LIN {X 0,Y 441.863,Z 860.022,A -85,B 0,C 180,E1 -9104.979,E2 -9104.979} C_VEL
LIN {X 0,Y 442.081,Z 852.631,A -85,B 0,C 180,E1 -9105.384,E2 -9105.384} C_VEL
LIN {X 0,Y 440.393,Z 839.206,A -85,B 0,C 180,E1 -9106.023,E2 -9106.023} C_VEL
LIN {X 0,Y 438.824,Z 827.47,A -85,B 0,C 180,E1 -9106.443,E2 -9106.443} C_VEL
LIN {X 0,Y 439.003,Z 818.523,A -85,B 0,C 180,E1 -9109.645,E2 -9109.645} C_VEL
LIN {X 0,Y 439.338,Z 809.24,A -85,B 0,C 180,E1 -9113.074,E2 -9113.074} C_VEL
LIN {X 0,Y 439.723,Z 800.458,A -85,B 0,C 180,E1 -9116.486,E2 -9116.486} C_VEL
LIN {X 0,Y 440.208,Z 792.815,A -85,B 0,C 180,E1 -9119.665,E2 -9119.665} C_VEL
LIN {X 0,Y 440.836,Z 785.884,A -85,B 0,C 180,E1 -9122.823,E2 -9122.823} C_VEL
LIN {X 0,Y 441.25,Z 781.634,A -85,B 0,C 180,E1 -9124.987,E2 -9124.987} C_VEL
LIN {X 0,Y 441.238,Z 777.8,A -85,B 0,C 180,E1 -9127.248,E2 -9127.248} C_VEL
LIN {X 0,Y 440.674,Z 774.022,A -85,B 0,C 180,E1 -9130.046,E2 -9130.046} C_VEL
LIN {X 0,Y 440.207,Z 771.332,A -85,B 0,C 180,E1 -9132.743,E2 -9132.743} C_VEL
LIN {X 0,Y 439.877,Z 769.661,A -85,B 0,C 180,E1 -9135.331,E2 -9135.331} C_VEL
LIN {X 0,Y 439.737,Z 768.806,A -85,B 0,C 180,E1 -9137.835,E2 -9137.835} C_VEL
LIN {X 0,Y 439.694,Z 768.625,A -85,B 0,C 180,E1 -9140.256,E2 -9140.256} C_VEL
LIN {X 0,Y 439.718,Z 769.039,A -85,B 0,C 180,E1 -9143.049,E2 -9143.049} C_VEL
LIN {X 0,Y 439.636,Z 770.08,A -85,B 0,C 180,E1 -9145.977,E2 -9145.977} C_VEL
LIN {X 0,Y 439.502,Z 771.14,A -85,B 0,C 180,E1 -9148.149,E2 -9148.149} C_VEL
LIN {X 0,Y 439.208,Z 773.033,A -85,B 0,C 180,E1 -9151.311,E2 -9151.311} C_VEL
LIN {X 0,Y 439.029,Z 775.128,A -85,B 0,C 180,E1 -9154.391,E2 -9154.391} C_VEL
LIN {X 0,Y 438.912,Z 777.387,A -85,B 0,C 180,E1 -9157.399,E2 -9157.399} C_VEL
LIN {X 0,Y 438.78,Z 779.764,A -85,B 0,C 180,E1 -9160.344,E2 -9160.344} C_VEL
LIN {X 0,Y 438.668,Z 782.635,A -85,B 0,C 180,E1 -9163.693,E2 -9163.693} C_VEL
LIN {X 0,Y 442.001,Z 795.437,A -85,B 0,C 180,E1 -9164.317,E2 -9164.317} C_VEL
LIN {X 0,Y 442.761,Z 800.41,A -85,B 0,C 180,E1 -9164.58,E2 -9164.58} C_VEL
LIN {X 0,Y 442.269,Z 812.861,A -85,B 0,C 180,E1 -9165.27,E2 -9165.27} C_VEL
LIN {X 0,Y 441.715,Z 823.88,A -85,B 0,C 180,E1 -9166.062,E2 -9166.062} C_VEL
LIN {X 0,Y 441.095,Z 835.387,A -85,B 0,C 180,E1 -9167.11,E2 -9167.11} C_VEL
LIN {X 0,Y 440.405,Z 845.56,A -85,B 0,C 180,E1 -9168.259,E2 -9168.259} C_VEL
LIN {X 0,Y 439.861,Z 855.273,A -85,B 0,C 180,E1 -9169.644,E2 -9169.644} C_VEL
LIN {X 0,Y 439.359,Z 863.095,A -85,B 0,C 180,E1 -9171.027,E2 -9171.027} C_VEL
LIN {X 0,Y 439.018,Z 868.375,A -85,B 0,C 180,E1 -9172.179,E2 -9172.179} C_VEL
LIN {X 0,Y 438.847,Z 873.537,A -85,B 0,C 180,E1 -9173.563,E2 -9173.563} C_VEL
LIN {X 0,Y 438.558,Z 877.539,A -85,B 0,C 180,E1 -9174.943,E2 -9174.943} C_VEL
LIN {X 0,Y 438.53,Z 880.466,A -85,B 0,C 180,E1 -9176.324,E2 -9176.324} C_VEL
LIN {X 0,Y 438.434,Z 881.88,A -85,B 0,C 180,E1 -9177.243,E2 -9177.243} C_VEL
LIN {X 0,Y 438.451,Z 882.856,A -85,B 0,C 180,E1 -9178.162,E2 -9178.162} C_VEL
LIN {X 0,Y 438.338,Z 883.651,A -85,B 0,C 180,E1 -9179.999,E2 -9179.999} C_VEL
LIN {X 0,Y 438.367,Z 883.419,A -85,B 0,C 180,E1 -9180.918,E2 -9180.918} C_VEL
LIN {X 0,Y 438.429,Z 882.781,A -85,B 0,C 180,E1 -9181.836,E2 -9181.836} C_VEL
LIN {X 0,Y 438.405,Z 881.756,A -85,B 0,C 180,E1 -9182.756,E2 -9182.756} C_VEL
LIN {X 0,Y 438.516,Z 880.324,A -85,B 0,C 180,E1 -9183.675,E2 -9183.675} C_VEL
LIN {X 0,Y 438.493,Z 877.344,A -85,B 0,C 180,E1 -9185.056,E2 -9185.056} C_VEL
LIN {X 0,Y 438.765,Z 873.305,A -85,B 0,C 180,E1 -9186.437,E2 -9186.437} C_VEL
LIN {X 0,Y 438.997,Z 867.096,A -85,B 0,C 180,E1 -9188.052,E2 -9188.052} C_VEL
LIN {X 0,Y 439.42,Z 860.319,A -85,B 0,C 180,E1 -9189.434,E2 -9189.434} C_VEL
LIN {X 0,Y 439.925,Z 851.912,A -85,B 0,C 180,E1 -9190.818,E2 -9190.818} C_VEL
LIN {X 0,Y 440.418,Z 843.258,A -85,B 0,C 180,E1 -9191.972,E2 -9191.972} C_VEL
LIN {X 0,Y 441.03,Z 833.231,A -85,B 0,C 180,E1 -9193.064,E2 -9193.064} C_VEL
LIN {X 0,Y 441.548,Z 822.138,A -85,B 0,C 180,E1 -9194.047,E2 -9194.047} C_VEL
LIN {X 0,Y 442.104,Z 810.557,A -85,B 0,C 180,E1 -9194.852,E2 -9194.852} C_VEL
LIN {X 0,Y 442.538,Z 799.996,A -85,B 0,C 180,E1 -9195.426,E2 -9195.426} C_VEL
LIN {X 0,Y 440.768,Z 790.018,A -85,B 0,C 180,E1 -9195.922,E2 -9195.922} C_VEL
LIN {X 0,Y 438.433,Z 780.272,A -85,B 0,C 180,E1 -9196.344,E2 -9196.344} C_VEL
LIN {X 0,Y 438.467,Z 776.8,A -85,B 0,C 180,E1 -9199.669,E2 -9199.669} C_VEL
LIN {X 0,Y 438.535,Z 773.779,A -85,B 0,C 180,E1 -9202.619,E2 -9202.619} C_VEL
LIN {X 0,Y 438.643,Z 770.171,A -85,B 0,C 180,E1 -9206.202,E2 -9206.202} C_VEL
LIN {X 0,Y 438.702,Z 766.841,A -85,B 0,C 180,E1 -9209.775,E2 -9209.775} C_VEL
LIN {X 0,Y 439.093,Z 766.791,A -85,B 0,C 180,E1 -9212.968,E2 -9212.968} C_VEL
LIN {X 0,Y 439.308,Z 766.762,A -85,B 0,C 180,E1 -9215.324,E2 -9215.324} C_VEL
LIN {X 0,Y 439.373,Z 766.754,A -85,B 0,C 180,E1 -9218.594,E2 -9218.594} C_VEL
LIN {X 0,Y 439.384,Z 766.754,A -85,B 0,C 180,E1 -9221.256,E2 -9221.256} C_VEL
LIN {X 0,Y 439.396,Z 766.751,A -85,B 0,C 180,E1 -9224.728,E2 -9224.728} C_VEL
LIN {X 0,Y 439.39,Z 766.752,A -85,B 0,C 180,E1 -9227.795,E2 -9227.795} C_VEL
LIN {X 0,Y 439.404,Z 766.749,A -85,B 0,C 180,E1 -9230.225,E2 -9230.225} C_VEL
LIN {X 0,Y 439.366,Z 766.755,A -85,B 0,C 180,E1 -9233.712,E2 -9233.712} C_VEL
LIN {X 0,Y 439.364,Z 766.756,A -85,B 0,C 180,E1 -9237.053,E2 -9237.053} C_VEL
LIN {X 0,Y 439.369,Z 766.754,A -85,B 0,C 180,E1 -9240.273,E2 -9240.273} C_VEL
LIN {X 0,Y 439.373,Z 766.757,A -85,B 0,C 180,E1 -9243.392,E2 -9243.392} C_VEL
LIN {X 0,Y 439.373,Z 766.752,A -85,B 0,C 180,E1 -9246.429,E2 -9246.429} C_VEL
LIN {X 0,Y 439.379,Z 766.755,A -85,B 0,C 180,E1 -9249.397,E2 -9249.397} C_VEL
LIN {X 0,Y 439.395,Z 766.75,A -85,B 0,C 180,E1 -9252.308,E2 -9252.308} C_VEL
LIN {X 0,Y 439.437,Z 766.745,A -85,B 0,C 180,E1 -9255.174,E2 -9255.174} C_VEL
LIN {X 0,Y 439.473,Z 766.743,A -85,B 0,C 180,E1 -9258.001,E2 -9258.001} C_VEL
LIN {X 0,Y 439.491,Z 766.742,A -85,B 0,C 180,E1 -9261.725,E2 -9261.725} C_VEL
LIN {X 0,Y 439.586,Z 766.725,A -85,B 0,C 180,E1 -9264.495,E2 -9264.495} C_VEL
LIN {X 0,Y 439.516,Z 766.732,A -85,B 0,C 180,E1 -9266.988,E2 -9266.988} C_VEL
LIN {X 0,Y 439.304,Z 766.763,A -85,B 0,C 180,E1 -9267.499,E2 -9267.499} C_VEL
LIN {X 0,Y 438.003,Z 766.928,A -85,B 0,C 180,E1 -9268.254,E2 -9268.254} C_VEL
LIN {X 0,Y 433.58,Z 767.48,A -85,B 0,C 180,E1 -9269.996,E2 -9269.996} C_VEL
LIN {X 0,Y 432.529,Z 767.604,A -85,B 0,C 180,E1 -9270.773,E2 -9270.773} C_VEL
LIN {X 0,Y 432.464,Z 767.611,A -85,B 0,C 180,E1 -9271.036,E2 -9271.036} C_VEL
LIN {X 0,Y 432.543,Z 767.601,A -85,B 0,C 180,E1 -9272.794,E2 -9272.794} C_VEL
LIN {X 0,Y 432.503,Z 767.609,A -85,B 0,C 180,E1 -9276.531,E2 -9276.531} C_VEL
LIN {X 0,Y 432.408,Z 767.618,A -85,B 0,C 180,E1 -9279.354,E2 -9279.354} C_VEL
LIN {X 0,Y 432.421,Z 767.618,A -85,B 0,C 180,E1 -9282.803,E2 -9282.803} C_VEL
LIN {X 0,Y 432.402,Z 767.625,A -85,B 0,C 180,E1 -9286.478,E2 -9286.478} C_VEL
LIN {X 0,Y 432.329,Z 767.63,A -85,B 0,C 180,E1 -9289.961,E2 -9289.961} C_VEL
LIN {X 0,Y 432.307,Z 767.633,A -85,B 0,C 180,E1 -9292.965,E2 -9292.965} C_VEL
LIN {X 0,Y 432.325,Z 767.631,A -85,B 0,C 180,E1 -9295.003,E2 -9295.003} C_VEL
LIN {X 0,Y 432.334,Z 767.63,A -85,B 0,C 180,E1 -9298.127,E2 -9298.127} C_VEL
LIN {X 0,Y 432.312,Z 767.632,A -85,B 0,C 180,E1 -9301.347,E2 -9301.347} C_VEL
LIN {X 0,Y 432.33,Z 767.634,A -85,B 0,C 180,E1 -9304.678,E2 -9304.678} C_VEL
LIN {X 0,Y 432.329,Z 767.63,A -85,B 0,C 180,E1 -9308.151,E2 -9308.151} C_VEL
LIN {X 0,Y 432.326,Z 767.631,A -85,B 0,C 180,E1 -9311.603,E2 -9311.603} C_VEL
LIN {X 0,Y 432.328,Z 767.631,A -85,B 0,C 180,E1 -9314.348,E2 -9314.348} C_VEL
LIN {X 0,Y 432.315,Z 767.637,A -85,B 0,C 180,E1 -9317.017,E2 -9317.017} C_VEL
LIN {X 0,Y 432.329,Z 767.631,A -85,B 0,C 180,E1 -9319.822,E2 -9319.822} C_VEL
LIN {X 0,Y 432.295,Z 767.638,A -85,B 0,C 180,E1 -9323.022,E2 -9323.022} C_VEL
LIN {X 0,Y 432.168,Z 767.654,A -85,B 0,C 180,E1 -9326.035,E2 -9326.035} C_VEL
LIN {X 0,Y 431.864,Z 767.69,A -85,B 0,C 180,E1 -9328.618,E2 -9328.618} C_VEL
LIN {X 0,Y 431.471,Z 767.743,A -85,B 0,C 180,E1 -9331.813,E2 -9331.813} C_VEL
LIN {X 0,Y 431.514,Z 769.976,A -85,B 0,C 180,E1 -9333.914,E2 -9333.914} C_VEL
LIN {X 0,Y 431.405,Z 773.326,A -85,B 0,C 180,E1 -9336.986,E2 -9336.986} C_VEL
LIN {X 0,Y 431.382,Z 776.555,A -85,B 0,C 180,E1 -9339.995,E2 -9339.995} C_VEL
LIN {X 0,Y 431.355,Z 780.414,A -85,B 0,C 180,E1 -9343.533,E2 -9343.533} C_VEL
LIN {X 0,Y 434.362,Z 793.612,A -85,B 0,C 180,E1 -9344.097,E2 -9344.097} C_VEL
LIN {X 0,Y 435.602,Z 801.29,A -85,B 0,C 180,E1 -9344.504,E2 -9344.504} C_VEL
LIN {X 0,Y 435.12,Z 812.506,A -85,B 0,C 180,E1 -9345.144,E2 -9345.144} C_VEL
LIN {X 0,Y 434.523,Z 823.742,A -85,B 0,C 180,E1 -9345.96,E2 -9345.96} C_VEL
LIN {X 0,Y 433.987,Z 835.113,A -85,B 0,C 180,E1 -9347.016,E2 -9347.016} C_VEL
LIN {X 0,Y 433.335,Z 844.381,A -85,B 0,C 180,E1 -9348.067,E2 -9348.067} C_VEL
LIN {X 0,Y 432.861,Z 852.9,A -85,B 0,C 180,E1 -9349.24,E2 -9349.24} C_VEL
LIN {X 0,Y 432.333,Z 861.184,A -85,B 0,C 180,E1 -9350.646,E2 -9350.646} C_VEL
LIN {X 0,Y 431.905,Z 867.856,A -85,B 0,C 180,E1 -9352.051,E2 -9352.051} C_VEL
LIN {X 0,Y 431.699,Z 873.179,A -85,B 0,C 180,E1 -9353.457,E2 -9353.457} C_VEL
LIN {X 0,Y 431.44,Z 877.326,A -85,B 0,C 180,E1 -9354.861,E2 -9354.861} C_VEL
LIN {X 0,Y 431.45,Z 880.397,A -85,B 0,C 180,E1 -9356.265,E2 -9356.265} C_VEL
LIN {X 0,Y 431.33,Z 881.916,A -85,B 0,C 180,E1 -9357.199,E2 -9357.199} C_VEL
LIN {X 0,Y 431.328,Z 882.978,A -85,B 0,C 180,E1 -9358.133,E2 -9358.133} C_VEL
LIN {X 0,Y 431.308,Z 883.654,A -85,B 0,C 180,E1 -9359.067,E2 -9359.067} C_VEL
LIN {X 0,Y 431.277,Z 883.943,A -85,B 0,C 180,E1 -9360.001,E2 -9360.001} C_VEL
LIN {X 0,Y 431.309,Z 883.789,A -85,B 0,C 180,E1 -9360.935,E2 -9360.935} C_VEL
LIN {X 0,Y 431.345,Z 883.232,A -85,B 0,C 180,E1 -9361.868,E2 -9361.868} C_VEL
LIN {X 0,Y 431.348,Z 882.291,A -85,B 0,C 180,E1 -9362.803,E2 -9362.803} C_VEL
LIN {X 0,Y 431.466,Z 880.928,A -85,B 0,C 180,E1 -9363.737,E2 -9363.737} C_VEL
LIN {X 0,Y 431.467,Z 878.071,A -85,B 0,C 180,E1 -9365.141,E2 -9365.141} C_VEL
LIN {X 0,Y 431.78,Z 874.144,A -85,B 0,C 180,E1 -9366.543,E2 -9366.543} C_VEL
LIN {X 0,Y 431.987,Z 869.057,A -85,B 0,C 180,E1 -9367.95,E2 -9367.95} C_VEL
LIN {X 0,Y 432.396,Z 862.638,A -85,B 0,C 180,E1 -9369.355,E2 -9369.355} C_VEL
LIN {X 0,Y 432.955,Z 854.665,A -85,B 0,C 180,E1 -9370.76,E2 -9370.76} C_VEL
LIN {X 0,Y 433.454,Z 846.49,A -85,B 0,C 180,E1 -9371.932,E2 -9371.932} C_VEL
LIN {X 0,Y 434.143,Z 836.441,A -85,B 0,C 180,E1 -9373.1,E2 -9373.1} C_VEL
LIN {X 0,Y 434.685,Z 825.348,A -85,B 0,C 180,E1 -9374.156,E2 -9374.156} C_VEL
LIN {X 0,Y 435.439,Z 812.658,A -85,B 0,C 180,E1 -9375.086,E2 -9375.086} C_VEL
LIN {X 0,Y 435.939,Z 801.427,A -85,B 0,C 180,E1 -9375.727,E2 -9375.727} C_VEL
LIN {X 0,Y 434.163,Z 791.998,A -85,B 0,C 180,E1 -9376.237,E2 -9376.237} C_VEL
LIN {X 0,Y 431.559,Z 782.504,A -85,B 0,C 180,E1 -9376.694,E2 -9376.694} C_VEL
LIN {X 0,Y 431.548,Z 778.931,A -85,B 0,C 180,E1 -9379.999,E2 -9379.999} C_VEL
LIN {X 0,Y 431.615,Z 775.631,A -85,B 0,C 180,E1 -9383.005,E2 -9383.005} C_VEL
LIN {X 0,Y 431.67,Z 772.181,A -85,B 0,C 180,E1 -9386.078,E2 -9386.078} C_VEL
LIN {X 0,Y 431.645,Z 768.422,A -85,B 0,C 180,E1 -9389.24,E2 -9389.24} C_VEL
LIN {X 0,Y 431.711,Z 767.713,A -85,B 0,C 180,E1 -9390.366,E2 -9390.366} C_VEL
LIN {X 0,Y 432.113,Z 767.663,A -85,B 0,C 180,E1 -9393.573,E2 -9393.573} C_VEL
LIN {X 0,Y 432.273,Z 767.639,A -85,B 0,C 180,E1 -9395.825,E2 -9395.825} C_VEL
LIN {X 0,Y 432.337,Z 767.632,A -85,B 0,C 180,E1 -9398.713,E2 -9398.713} C_VEL
LIN {X 0,Y 432.329,Z 767.631,A -85,B 0,C 180,E1 -9401.799,E2 -9401.799} C_VEL
LIN {X 0,Y 432.338,Z 767.631,A -85,B 0,C 180,E1 -9404.348,E2 -9404.348} C_VEL
LIN {X 0,Y 432.382,Z 767.68,A -85,B 0,C 180,E1 -9407.817,E2 -9407.817} C_VEL
LIN {X 0,Y 433.57,Z 774.337,A -85,B 0,C 180,E1 -9411.084,E2 -9411.084} C_VEL
LIN {X 0,Y 434.286,Z 778.889,A -85,B 0,C 180,E1 -9413.218,E2 -9413.218} C_VEL
LIN {X 0,Y 434.361,Z 782.778,A -85,B 0,C 180,E1 -9414.943,E2 -9414.943} C_VEL
LIN {X 0,Y 433.81,Z 790.498,A -85,B 0,C 180,E1 -9418.229,E2 -9418.229} C_VEL
LIN {X 0,Y 433.312,Z 797.589,A -85,B 0,C 180,E1 -9421.146,E2 -9421.146} C_VEL
LIN {X 0,Y 432.793,Z 805.999,A -85,B 0,C 180,E1 -9424.512,E2 -9424.512} C_VEL
LIN {X 0,Y 432.309,Z 815.073,A -85,B 0,C 180,E1 -9428.043,E2 -9428.043} C_VEL
LIN {X 0,Y 432,Z 822.85,A -85,B 0,C 180,E1 -9431.012,E2 -9431.012} C_VEL
LIN {X 0,Y 431.769,Z 829.127,A -85,B 0,C 180,E1 -9433.372,E2 -9433.372} C_VEL
LIN {X 0,Y 433.924,Z 843.779,A -85,B 0,C 180,E1 -9433.915,E2 -9433.915} C_VEL
LIN {X 0,Y 435.32,Z 855.22,A -85,B 0,C 180,E1 -9434.491,E2 -9434.491} C_VEL
LIN {X 0,Y 434.594,Z 867.79,A -85,B 0,C 180,E1 -9435.244,E2 -9435.244} C_VEL
LIN {X 0,Y 433.967,Z 879.201,A -85,B 0,C 180,E1 -9436.128,E2 -9436.128} C_VEL
LIN {X 0,Y 433.304,Z 890.451,A -85,B 0,C 180,E1 -9437.233,E2 -9437.233} C_VEL
LIN {X 0,Y 432.665,Z 901.007,A -85,B 0,C 180,E1 -9438.522,E2 -9438.522} C_VEL
LIN {X 0,Y 432.12,Z 910.17,A -85,B 0,C 180,E1 -9439.931,E2 -9439.931} C_VEL
LIN {X 0,Y 431.75,Z 917.565,A -85,B 0,C 180,E1 -9441.34,E2 -9441.34} C_VEL
LIN {X 0,Y 431.538,Z 922.578,A -85,B 0,C 180,E1 -9442.514,E2 -9442.514} C_VEL
LIN {X 0,Y 431.329,Z 927.577,A -85,B 0,C 180,E1 -9443.967,E2 -9443.967} C_VEL
LIN {X 0,Y 431.292,Z 931.148,A -85,B 0,C 180,E1 -9445.327,E2 -9445.327} C_VEL
LIN {X 0,Y 431.235,Z 933.056,A -85,B 0,C 180,E1 -9446.262,E2 -9446.262} C_VEL
LIN {X 0,Y 431.287,Z 934.499,A -85,B 0,C 180,E1 -9447.198,E2 -9447.198} C_VEL
LIN {X 0,Y 431.273,Z 935.505,A -85,B 0,C 180,E1 -9448.132,E2 -9448.132} C_VEL
LIN {X 0,Y 431.29,Z 936.109,A -85,B 0,C 180,E1 -9449.066,E2 -9449.066} C_VEL
LIN {X 0,Y 431.278,Z 936.308,A -85,B 0,C 180,E1 -9450,E2 -9450} C_VEL
LIN {X 0,Y 431.29,Z 936.059,A -85,B 0,C 180,E1 -9450.934,E2 -9450.934} C_VEL
LIN {X 0,Y 431.273,Z 935.396,A -85,B 0,C 180,E1 -9451.868,E2 -9451.868} C_VEL
LIN {X 0,Y 431.293,Z 934.326,A -85,B 0,C 180,E1 -9452.802,E2 -9452.802} C_VEL
LIN {X 0,Y 431.26,Z 932.833,A -85,B 0,C 180,E1 -9453.738,E2 -9453.738} C_VEL
LIN {X 0,Y 431.374,Z 929.731,A -85,B 0,C 180,E1 -9455.141,E2 -9455.141} C_VEL
LIN {X 0,Y 431.388,Z 925.534,A -85,B 0,C 180,E1 -9456.548,E2 -9456.548} C_VEL
LIN {X 0,Y 431.643,Z 919.105,A -85,B 0,C 180,E1 -9458.191,E2 -9458.191} C_VEL
LIN {X 0,Y 431.958,Z 912.134,A -85,B 0,C 180,E1 -9459.6,E2 -9459.6} C_VEL
LIN {X 0,Y 432.421,Z 903.502,A -85,B 0,C 180,E1 -9461.009,E2 -9461.009} C_VEL
LIN {X 0,Y 432.962,Z 894.653,A -85,B 0,C 180,E1 -9462.182,E2 -9462.182} C_VEL
LIN {X 0,Y 433.62,Z 883.449,A -85,B 0,C 180,E1 -9463.394,E2 -9463.394} C_VEL
LIN {X 0,Y 434.284,Z 871.69,A -85,B 0,C 180,E1 -9464.407,E2 -9464.407} C_VEL
LIN {X 0,Y 434.987,Z 859.664,A -85,B 0,C 180,E1 -9465.221,E2 -9465.221} C_VEL
LIN {X 0,Y 435.171,Z 853.459,A -85,B 0,C 180,E1 -9465.575,E2 -9465.575} C_VEL
LIN {X 0,Y 433.634,Z 840.529,A -85,B 0,C 180,E1 -9466.24,E2 -9466.24} C_VEL
LIN {X 0,Y 431.764,Z 826.891,A -85,B 0,C 180,E1 -9466.769,E2 -9466.769} C_VEL
LIN {X 0,Y 431.981,Z 816.805,A -85,B 0,C 180,E1 -9470.474,E2 -9470.474} C_VEL
LIN {X 0,Y 432.314,Z 808.928,A -85,B 0,C 180,E1 -9473.471,E2 -9473.471} C_VEL
LIN {X 0,Y 432.701,Z 800.839,A -85,B 0,C 180,E1 -9476.706,E2 -9476.706} C_VEL
LIN {X 0,Y 433.171,Z 793.917,A -85,B 0,C 180,E1 -9479.66,E2 -9479.66} C_VEL
LIN {X 0,Y 433.807,Z 787.598,A -85,B 0,C 180,E1 -9482.6,E2 -9482.6} C_VEL
LIN {X 0,Y 434.279,Z 782.849,A -85,B 0,C 180,E1 -9485.065,E2 -9485.065} C_VEL
LIN {X 0,Y 434.314,Z 779.975,A -85,B 0,C 180,E1 -9486.779,E2 -9486.779} C_VEL
LIN {X 0,Y 433.911,Z 776.606,A -85,B 0,C 180,E1 -9489.174,E2 -9489.174} C_VEL
LIN {X 0,Y 433.449,Z 773.755,A -85,B 0,C 180,E1 -9491.767,E2 -9491.767} C_VEL
LIN {X 0,Y 433.087,Z 771.695,A -85,B 0,C 180,E1 -9494.436,E2 -9494.436} C_VEL
LIN {X 0,Y 432.835,Z 770.539,A -85,B 0,C 180,E1 -9497.002,E2 -9497.002} C_VEL
LIN {X 0,Y 432.741,Z 770.076,A -85,B 0,C 180,E1 -9499.757,E2 -9499.757} C_VEL
LIN {X 0,Y 432.761,Z 770.401,A -85,B 0,C 180,E1 -9503.066,E2 -9503.066} C_VEL
LIN {X 0,Y 432.669,Z 771.316,A -85,B 0,C 180,E1 -9505.936,E2 -9505.936} C_VEL
LIN {X 0,Y 432.425,Z 772.622,A -85,B 0,C 180,E1 -9508.662,E2 -9508.662} C_VEL
LIN {X 0,Y 432.164,Z 774.491,A -85,B 0,C 180,E1 -9511.86,E2 -9511.86} C_VEL
LIN {X 0,Y 431.973,Z 776.592,A -85,B 0,C 180,E1 -9514.975,E2 -9514.975} C_VEL
LIN {X 0,Y 431.865,Z 778.876,A -85,B 0,C 180,E1 -9518.064,E2 -9518.064} C_VEL
LIN {X 0,Y 431.72,Z 781.225,A -85,B 0,C 180,E1 -9520.998,E2 -9520.998} C_VEL
LIN {X 0,Y 431.647,Z 783.41,A -85,B 0,C 180,E1 -9523.394,E2 -9523.394} C_VEL
LIN {X 0,Y 434.777,Z 794.715,A -85,B 0,C 180,E1 -9523.957,E2 -9523.957} C_VEL
LIN {X 0,Y 435.993,Z 801.499,A -85,B 0,C 180,E1 -9524.335,E2 -9524.335} C_VEL
LIN {X 0,Y 435.452,Z 813.692,A -85,B 0,C 180,E1 -9525.034,E2 -9525.034} C_VEL
LIN {X 0,Y 434.853,Z 824.832,A -85,B 0,C 180,E1 -9525.862,E2 -9525.862} C_VEL
LIN {X 0,Y 434.203,Z 835.954,A -85,B 0,C 180,E1 -9526.902,E2 -9526.902} C_VEL
LIN {X 0,Y 433.482,Z 846.108,A -85,B 0,C 180,E1 -9528.069,E2 -9528.069} C_VEL
LIN {X 0,Y 432.909,Z 855.81,A -85,B 0,C 180,E1 -9529.476,E2 -9529.476} C_VEL
LIN {X 0,Y 432.371,Z 863.624,A -85,B 0,C 180,E1 -9530.88,E2 -9530.88} C_VEL
LIN {X 0,Y 432.005,Z 868.899,A -85,B 0,C 180,E1 -9532.051,E2 -9532.051} C_VEL
LIN {X 0,Y 431.81,Z 874.036,A -85,B 0,C 180,E1 -9533.457,E2 -9533.457} C_VEL
LIN {X 0,Y 431.493,Z 878.019,A -85,B 0,C 180,E1 -9534.86,E2 -9534.86} C_VEL
LIN {X 0,Y 431.474,Z 880.929,A -85,B 0,C 180,E1 -9536.263,E2 -9536.263} C_VEL
LIN {X 0,Y 431.367,Z 882.334,A -85,B 0,C 180,E1 -9537.197,E2 -9537.197} C_VEL
LIN {X 0,Y 431.378,Z 883.302,A -85,B 0,C 180,E1 -9538.132,E2 -9538.132} C_VEL
LIN {X 0,Y 431.277,Z 884.085,A -85,B 0,C 180,E1 -9539.999,E2 -9539.999} C_VEL
LIN {X 0,Y 431.309,Z 883.843,A -85,B 0,C 180,E1 -9540.933,E2 -9540.933} C_VEL
LIN {X 0,Y 431.343,Z 883.195,A -85,B 0,C 180,E1 -9541.866,E2 -9541.866} C_VEL
LIN {X 0,Y 431.339,Z 882.159,A -85,B 0,C 180,E1 -9542.801,E2 -9542.801} C_VEL
LIN {X 0,Y 431.456,Z 880.713,A -85,B 0,C 180,E1 -9543.735,E2 -9543.735} C_VEL
LIN {X 0,Y 431.436,Z 877.712,A -85,B 0,C 180,E1 -9545.139,E2 -9545.139} C_VEL
LIN {X 0,Y 431.683,Z 873.016,A -85,B 0,C 180,E1 -9546.728,E2 -9546.728} C_VEL
LIN {X 0,Y 432.065,Z 866.374,A -85,B 0,C 180,E1 -9548.417,E2 -9548.417} C_VEL
LIN {X 0,Y 432.493,Z 859.325,A -85,B 0,C 180,E1 -9549.823,E2 -9549.823} C_VEL
LIN {X 0,Y 433.005,Z 850.503,A -85,B 0,C 180,E1 -9551.23,E2 -9551.23} C_VEL
LIN {X 0,Y 433.707,Z 840.507,A -85,B 0,C 180,E1 -9552.516,E2 -9552.516} C_VEL
LIN {X 0,Y 434.36,Z 829.162,A -85,B 0,C 180,E1 -9553.677,E2 -9553.677} C_VEL
LIN {X 0,Y 434.894,Z 817.59,A -85,B 0,C 180,E1 -9554.625,E2 -9554.625} C_VEL
LIN {X 0,Y 435.475,Z 805.595,A -85,B 0,C 180,E1 -9555.382,E2 -9555.382} C_VEL
LIN {X 0,Y 435.531,Z 799.942,A -85,B 0,C 180,E1 -9555.68,E2 -9555.68} C_VEL
LIN {X 0,Y 433.439,Z 789.306,A -85,B 0,C 180,E1 -9556.218,E2 -9556.218} C_VEL
LIN {X 0,Y 431.364,Z 780.619,A -85,B 0,C 180,E1 -9556.591,E2 -9556.591} C_VEL
LIN {X 0,Y 431.392,Z 777.094,A -85,B 0,C 180,E1 -9560.005,E2 -9560.005} C_VEL
LIN {X 0,Y 431.491,Z 774.016,A -85,B 0,C 180,E1 -9563.01,E2 -9563.01} C_VEL
LIN {X 0,Y 431.582,Z 770.613,A -85,B 0,C 180,E1 -9566.409,E2 -9566.409} C_VEL
LIN {X 0,Y 431.589,Z 767.837,A -85,B 0,C 180,E1 -9569.242,E2 -9569.242} C_VEL
LIN {X 0,Y 431.984,Z 767.679,A -85,B 0,C 180,E1 -9572.47,E2 -9572.47} C_VEL
LIN {X 0,Y 432.26,Z 767.64,A -85,B 0,C 180,E1 -9575.616,E2 -9575.616} C_VEL
LIN {X 0,Y 432.337,Z 767.632,A -85,B 0,C 180,E1 -9578.714,E2 -9578.714} C_VEL
LIN {X 0,Y 432.329,Z 767.631,A -85,B 0,C 180,E1 -9581.796,E2 -9581.796} C_VEL
LIN {X 0,Y 432.328,Z 767.631,A -85,B 0,C 180,E1 -9584.346,E2 -9584.346} C_VEL
LIN {X 0,Y 432.315,Z 767.636,A -85,B 0,C 180,E1 -9587.015,E2 -9587.015} C_VEL
LIN {X 0,Y 432.327,Z 767.631,A -85,B 0,C 180,E1 -9589.82,E2 -9589.82} C_VEL
LIN {X 0,Y 432.299,Z 767.637,A -85,B 0,C 180,E1 -9593.021,E2 -9593.021} C_VEL
LIN {X 0,Y 432.35,Z 767.628,A -85,B 0,C 180,E1 -9595.996,E2 -9595.996} C_VEL
LIN {X 0,Y 432.338,Z 767.633,A -85,B 0,C 180,E1 -9599.489,E2 -9599.489} C_VEL
LIN {X 0,Y 432.339,Z 767.63,A -85,B 0,C 180,E1 -9601.874,E2 -9601.874} C_VEL
LIN {X 0,Y 432.368,Z 767.63,A -85,B 0,C 180,E1 -9605.538,E2 -9605.538} C_VEL
LIN {X 0,Y 432.341,Z 767.629,A -85,B 0,C 180,E1 -9609.045,E2 -9609.045} C_VEL
LIN {X 0,Y 432.351,Z 767.629,A -85,B 0,C 180,E1 -9612.01,E2 -9612.01} C_VEL
LIN {X 0,Y 432.385,Z 767.622,A -85,B 0,C 180,E1 -9614.926,E2 -9614.926} C_VEL
LIN {X 0,Y 432.449,Z 767.62,A -85,B 0,C 180,E1 -9617.803,E2 -9617.803} C_VEL
LIN {X 0,Y 432.451,Z 767.617,A -85,B 0,C 180,E1 -9621.589,E2 -9621.589} C_VEL
LIN {X 0,Y 432.541,Z 767.603,A -85,B 0,C 180,E1 -9624.405,E2 -9624.405} C_VEL
LIN {X 0,Y 432.584,Z 767.602,A -85,B 0,C 180,E1 -9628.138,E2 -9628.138} C_VEL
LIN {X 0,Y 432.609,Z 767.601,A -85,B 0,C 180,E1 -9630,E2 -9630} C_VEL
LIN {X 0,Y 432.464,Z 767.611,A -85,B 0,C 180,E1 -9631.036,E2 -9631.036} C_VEL
LIN {X 0,Y 431.824,Z 767.697,A -85,B 0,C 180,E1 -9631.813,E2 -9631.813} C_VEL
LIN {X 0,Y 428.891,Z 768.056,A -85,B 0,C 180,E1 -9633.073,E2 -9633.073} C_VEL
LIN {X 0,Y 426.426,Z 768.371,A -85,B 0,C 180,E1 -9634.091,E2 -9634.091} C_VEL
LIN {X 0,Y 425.431,Z 768.488,A -85,B 0,C 180,E1 -9634.879,E2 -9634.879} C_VEL
LIN {X 0,Y 425.387,Z 768.492,A -85,B 0,C 180,E1 -9635.145,E2 -9635.145} C_VEL
LIN {X 0,Y 425.47,Z 768.484,A -85,B 0,C 180,E1 -9637.664,E2 -9637.664} C_VEL
LIN {X 0,Y 425.331,Z 768.504,A -85,B 0,C 180,E1 -9640.472,E2 -9640.472} C_VEL
LIN {X 0,Y 425.355,Z 768.497,A -85,B 0,C 180,E1 -9643.375,E2 -9643.375} C_VEL
LIN {X 0,Y 425.351,Z 768.502,A -85,B 0,C 180,E1 -9646.605,E2 -9646.605} C_VEL
LIN {X 0,Y 425.319,Z 768.502,A -85,B 0,C 180,E1 -9649.636,E2 -9649.636} C_VEL
LIN {X 0,Y 425.279,Z 768.512,A -85,B 0,C 180,E1 -9652.339,E2 -9652.339} C_VEL
LIN {X 0,Y 425.308,Z 768.509,A -85,B 0,C 180,E1 -9654.657,E2 -9654.657} C_VEL
LIN {X 0,Y 425.26,Z 768.51,A -85,B 0,C 180,E1 -9657.564,E2 -9657.564} C_VEL
LIN {X 0,Y 425.282,Z 768.512,A -85,B 0,C 180,E1 -9660.762,E2 -9660.762} C_VEL
LIN {X 0,Y 425.302,Z 768.506,A -85,B 0,C 180,E1 -9664.288,E2 -9664.288} C_VEL
LIN {X 0,Y 425.272,Z 768.509,A -85,B 0,C 180,E1 -9667.695,E2 -9667.695} C_VEL
LIN {X 0,Y 425.273,Z 768.511,A -85,B 0,C 180,E1 -9670.521,E2 -9670.521} C_VEL
LIN {X 0,Y 425.251,Z 768.513,A -85,B 0,C 180,E1 -9673.352,E2 -9673.352} C_VEL
LIN {X 0,Y 425.252,Z 768.513,A -85,B 0,C 180,E1 -9676.65,E2 -9676.65} C_VEL
LIN {X 0,Y 425.282,Z 768.509,A -85,B 0,C 180,E1 -9679.874,E2 -9679.874} C_VEL
LIN {X 0,Y 425.271,Z 768.51,A -85,B 0,C 180,E1 -9682.49,E2 -9682.49} C_VEL
LIN {X 0,Y 425.156,Z 768.528,A -85,B 0,C 180,E1 -9685.805,E2 -9685.805} C_VEL
LIN {X 0,Y 424.906,Z 768.559,A -85,B 0,C 180,E1 -9688.044,E2 -9688.044} C_VEL
LIN {X 0,Y 424.482,Z 768.613,A -85,B 0,C 180,E1 -9691.343,E2 -9691.343} C_VEL
LIN {X 0,Y 424.411,Z 768.972,A -85,B 0,C 180,E1 -9692.378,E2 -9692.378} C_VEL
LIN {X 0,Y 424.376,Z 772.446,A -85,B 0,C 180,E1 -9695.623,E2 -9695.623} C_VEL
LIN {X 0,Y 424.348,Z 775.701,A -85,B 0,C 180,E1 -9698.633,E2 -9698.633} C_VEL
LIN {X 0,Y 424.274,Z 778.978,A -85,B 0,C 180,E1 -9701.657,E2 -9701.657} C_VEL
LIN {X 0,Y 424.294,Z 780.917,A -85,B 0,C 180,E1 -9703.291,E2 -9703.291} C_VEL
LIN {X 0,Y 427.445,Z 794.465,A -85,B 0,C 180,E1 -9703.888,E2 -9703.888} C_VEL
LIN {X 0,Y 428.712,Z 802.123,A -85,B 0,C 180,E1 -9704.303,E2 -9704.303} C_VEL
LIN {X 0,Y 428.163,Z 814.221,A -85,B 0,C 180,E1 -9705.019,E2 -9705.019} C_VEL
LIN {X 0,Y 427.556,Z 825.563,A -85,B 0,C 180,E1 -9705.889,E2 -9705.889} C_VEL
LIN {X 0,Y 426.937,Z 837.439,A -85,B 0,C 180,E1 -9707.04,E2 -9707.04} C_VEL
LIN {X 0,Y 426.275,Z 846.365,A -85,B 0,C 180,E1 -9708.108,E2 -9708.108} C_VEL
LIN {X 0,Y 425.669,Z 856.043,A -85,B 0,C 180,E1 -9709.537,E2 -9709.537} C_VEL
LIN {X 0,Y 425.182,Z 863.838,A -85,B 0,C 180,E1 -9710.967,E2 -9710.967} C_VEL
LIN {X 0,Y 424.753,Z 870.056,A -85,B 0,C 180,E1 -9712.395,E2 -9712.395} C_VEL
LIN {X 0,Y 424.629,Z 874.991,A -85,B 0,C 180,E1 -9713.825,E2 -9713.825} C_VEL
LIN {X 0,Y 424.316,Z 878.801,A -85,B 0,C 180,E1 -9715.251,E2 -9715.251} C_VEL
LIN {X 0,Y 424.372,Z 880.757,A -85,B 0,C 180,E1 -9716.203,E2 -9716.203} C_VEL
LIN {X 0,Y 424.268,Z 882.297,A -85,B 0,C 180,E1 -9717.153,E2 -9717.153} C_VEL
LIN {X 0,Y 424.246,Z 883.374,A -85,B 0,C 180,E1 -9718.102,E2 -9718.102} C_VEL
LIN {X 0,Y 424.203,Z 884.365,A -85,B 0,C 180,E1 -9720.001,E2 -9720.001} C_VEL
LIN {X 0,Y 424.252,Z 884.227,A -85,B 0,C 180,E1 -9720.95,E2 -9720.95} C_VEL
LIN {X 0,Y 424.285,Z 882.75,A -85,B 0,C 180,E1 -9722.849,E2 -9722.849} C_VEL
LIN {X 0,Y 424.409,Z 881.4,A -85,B 0,C 180,E1 -9723.799,E2 -9723.799} C_VEL
LIN {X 0,Y 424.41,Z 878.554,A -85,B 0,C 180,E1 -9725.227,E2 -9725.227} C_VEL
LIN {X 0,Y 424.748,Z 873.863,A -85,B 0,C 180,E1 -9726.889,E2 -9726.889} C_VEL
LIN {X 0,Y 425.109,Z 867.593,A -85,B 0,C 180,E1 -9728.558,E2 -9728.558} C_VEL
LIN {X 0,Y 425.587,Z 860.68,A -85,B 0,C 180,E1 -9729.986,E2 -9729.986} C_VEL
LIN {X 0,Y 426.235,Z 852.124,A -85,B 0,C 180,E1 -9731.413,E2 -9731.413} C_VEL
LIN {X 0,Y 426.833,Z 843.37,A -85,B 0,C 180,E1 -9732.602,E2 -9732.602} C_VEL
LIN {X 0,Y 427.508,Z 832.787,A -85,B 0,C 180,E1 -9733.764,E2 -9733.764} C_VEL
LIN {X 0,Y 428.159,Z 821.761,A -85,B 0,C 180,E1 -9734.74,E2 -9734.74} C_VEL
LIN {X 0,Y 428.837,Z 809.797,A -85,B 0,C 180,E1 -9735.568,E2 -9735.568} C_VEL
LIN {X 0,Y 429.052,Z 801.326,A -85,B 0,C 180,E1 -9736.047,E2 -9736.047} C_VEL
LIN {X 0,Y 426.388,Z 789.477,A -85,B 0,C 180,E1 -9736.709,E2 -9736.709} C_VEL
LIN {X 0,Y 424.506,Z 783.023,A -85,B 0,C 180,E1 -9737.053,E2 -9737.053} C_VEL
LIN {X 0,Y 424.57,Z 780.552,A -85,B 0,C 180,E1 -9739.346,E2 -9739.346} C_VEL
LIN {X 0,Y 424.614,Z 776.144,A -85,B 0,C 180,E1 -9743.406,E2 -9743.406} C_VEL
LIN {X 0,Y 424.629,Z 772.447,A -85,B 0,C 180,E1 -9746.651,E2 -9746.651} C_VEL
LIN {X 0,Y 424.608,Z 768.846,A -85,B 0,C 180,E1 -9749.773,E2 -9749.773} C_VEL
LIN {X 0,Y 424.94,Z 768.556,A -85,B 0,C 180,E1 -9752.49,E2 -9752.49} C_VEL
LIN {X 0,Y 425.222,Z 768.521,A -85,B 0,C 180,E1 -9755.344,E2 -9755.344} C_VEL
LIN {X 0,Y 425.279,Z 768.511,A -85,B 0,C 180,E1 -9757.695,E2 -9757.695} C_VEL
LIN {X 0,Y 425.281,Z 768.511,A -85,B 0,C 180,E1 -9760.52,E2 -9760.52} C_VEL
LIN {X 0,Y 425.265,Z 768.511,A -85,B 0,C 180,E1 -9763.956,E2 -9763.956} C_VEL
LIN {X 0,Y 425.35,Z 768.602,A -85,B 0,C 180,E1 -9767.559,E2 -9767.559} C_VEL
LIN {X 0,Y 426.66,Z 776.009,A -85,B 0,C 180,E1 -9771.249,E2 -9771.249} C_VEL
LIN {X 0,Y 427.399,Z 781.207,A -85,B 0,C 180,E1 -9773.703,E2 -9773.703} C_VEL
LIN {X 0,Y 427.159,Z 786.355,A -85,B 0,C 180,E1 -9775.986,E2 -9775.986} C_VEL
LIN {X 0,Y 426.583,Z 794.08,A -85,B 0,C 180,E1 -9779.287,E2 -9779.287} C_VEL
LIN {X 0,Y 426.031,Z 801.823,A -85,B 0,C 180,E1 -9782.49,E2 -9782.49} C_VEL
LIN {X 0,Y 425.58,Z 809.567,A -85,B 0,C 180,E1 -9785.616,E2 -9785.616} C_VEL
LIN {X 0,Y 425.114,Z 818.616,A -85,B 0,C 180,E1 -9789.18,E2 -9789.18} C_VEL
LIN {X 0,Y 424.784,Z 826.371,A -85,B 0,C 180,E1 -9792.177,E2 -9792.177} C_VEL
LIN {X 0,Y 424.701,Z 828.822,A -85,B 0,C 180,E1 -9793.117,E2 -9793.117} C_VEL
LIN {X 0,Y 426.821,Z 842.833,A -85,B 0,C 180,E1 -9793.636,E2 -9793.636} C_VEL
LIN {X 0,Y 428.394,Z 855.579,A -85,B 0,C 180,E1 -9794.295,E2 -9794.295} C_VEL
LIN {X 0,Y 427.705,Z 867.106,A -85,B 0,C 180,E1 -9795.001,E2 -9795.001} C_VEL
LIN {X 0,Y 426.983,Z 879.088,A -85,B 0,C 180,E1 -9795.944,E2 -9795.944} C_VEL
LIN {X 0,Y 426.351,Z 889.856,A -85,B 0,C 180,E1 -9797.021,E2 -9797.021} C_VEL
LIN {X 0,Y 425.665,Z 900.446,A -85,B 0,C 180,E1 -9798.331,E2 -9798.331} C_VEL
LIN {X 0,Y 425.079,Z 909.641,A -85,B 0,C 180,E1 -9799.762,E2 -9799.762} C_VEL
LIN {X 0,Y 424.696,Z 917.06,A -85,B 0,C 180,E1 -9801.195,E2 -9801.195} C_VEL
LIN {X 0,Y 424.408,Z 923.864,A -85,B 0,C 180,E1 -9802.866,E2 -9802.866} C_VEL
LIN {X 0,Y 424.246,Z 928.339,A -85,B 0,C 180,E1 -9804.296,E2 -9804.296} C_VEL
LIN {X 0,Y 424.228,Z 930.696,A -85,B 0,C 180,E1 -9805.249,E2 -9805.249} C_VEL
LIN {X 0,Y 424.143,Z 932.608,A -85,B 0,C 180,E1 -9806.2,E2 -9806.2} C_VEL
LIN {X 0,Y 424.2,Z 934.062,A -85,B 0,C 180,E1 -9807.151,E2 -9807.151} C_VEL
LIN {X 0,Y 424.195,Z 935.071,A -85,B 0,C 180,E1 -9808.101,E2 -9808.101} C_VEL
LIN {X 0,Y 424.202,Z 935.676,A -85,B 0,C 180,E1 -9809.051,E2 -9809.051} C_VEL
LIN {X 0,Y 424.22,Z 935.878,A -85,B 0,C 180,E1 -9810,E2 -9810} C_VEL
LIN {X 0,Y 424.202,Z 935.628,A -85,B 0,C 180,E1 -9810.949,E2 -9810.949} C_VEL
LIN {X 0,Y 424.196,Z 934.958,A -85,B 0,C 180,E1 -9811.899,E2 -9811.899} C_VEL
LIN {X 0,Y 424.225,Z 933.887,A -85,B 0,C 180,E1 -9812.849,E2 -9812.849} C_VEL
LIN {X 0,Y 424.165,Z 932.391,A -85,B 0,C 180,E1 -9813.8,E2 -9813.8} C_VEL
LIN {X 0,Y 424.284,Z 929.286,A -85,B 0,C 180,E1 -9815.227,E2 -9815.227} C_VEL
LIN {X 0,Y 424.311,Z 925.094,A -85,B 0,C 180,E1 -9816.658,E2 -9816.658} C_VEL
LIN {X 0,Y 424.573,Z 918.673,A -85,B 0,C 180,E1 -9818.328,E2 -9818.328} C_VEL
LIN {X 0,Y 424.922,Z 911.692,A -85,B 0,C 180,E1 -9819.761,E2 -9819.761} C_VEL
LIN {X 0,Y 425.422,Z 903.057,A -85,B 0,C 180,E1 -9821.193,E2 -9821.193} C_VEL
LIN {X 0,Y 425.959,Z 894.204,A -85,B 0,C 180,E1 -9822.386,E2 -9822.386} C_VEL
LIN {X 0,Y 426.666,Z 882.945,A -85,B 0,C 180,E1 -9823.627,E2 -9823.627} C_VEL
LIN {X 0,Y 427.395,Z 871.424,A -85,B 0,C 180,E1 -9824.645,E2 -9824.645} C_VEL
LIN {X 0,Y 428.153,Z 859.579,A -85,B 0,C 180,E1 -9825.47,E2 -9825.47} C_VEL
LIN {X 0,Y 428.167,Z 853.47,A -85,B 0,C 180,E1 -9825.836,E2 -9825.836} C_VEL
LIN {X 0,Y 426.754,Z 840.706,A -85,B 0,C 180,E1 -9826.516,E2 -9826.516} C_VEL
LIN {X 0,Y 425.004,Z 828.524,A -85,B 0,C 180,E1 -9827.019,E2 -9827.019} C_VEL
LIN {X 0,Y 424.674,Z 826.342,A -85,B 0,C 180,E1 -9827.102,E2 -9827.102} C_VEL
LIN {X 0,Y 424.95,Z 816.451,A -85,B 0,C 180,E1 -9830.829,E2 -9830.829} C_VEL
LIN {X 0,Y 425.3,Z 808.648,A -85,B 0,C 180,E1 -9833.882,E2 -9833.882} C_VEL
LIN {X 0,Y 425.708,Z 801.23,A -85,B 0,C 180,E1 -9836.938,E2 -9836.938} C_VEL
LIN {X 0,Y 426.238,Z 793.87,A -85,B 0,C 180,E1 -9840.192,E2 -9840.192} C_VEL
LIN {X 0,Y 426.998,Z 787.174,A -85,B 0,C 180,E1 -9843.462,E2 -9843.462} C_VEL
LIN {X 0,Y 427.323,Z 784.089,A -85,B 0,C 180,E1 -9845.144,E2 -9845.144} C_VEL
LIN {X 0,Y 427.404,Z 782.128,A -85,B 0,C 180,E1 -9846.318,E2 -9846.318} C_VEL
LIN {X 0,Y 427.038,Z 778.692,A -85,B 0,C 180,E1 -9848.711,E2 -9848.711} C_VEL
LIN {X 0,Y 426.607,Z 775.824,A -85,B 0,C 180,E1 -9851.221,E2 -9851.221} C_VEL
LIN {X 0,Y 426.227,Z 773.65,A -85,B 0,C 180,E1 -9853.831,E2 -9853.831} C_VEL
LIN {X 0,Y 425.911,Z 772.232,A -85,B 0,C 180,E1 -9856.556,E2 -9856.556} C_VEL
LIN {X 0,Y 425.81,Z 771.567,A -85,B 0,C 180,E1 -9859.397,E2 -9859.397} C_VEL
LIN {X 0,Y 425.776,Z 771.661,A -85,B 0,C 180,E1 -9862.402,E2 -9862.402} C_VEL
LIN {X 0,Y 425.744,Z 772.189,A -85,B 0,C 180,E1 -9864.706,E2 -9864.706} C_VEL
LIN {X 0,Y 425.581,Z 773.208,A -85,B 0,C 180,E1 -9867.375,E2 -9867.375} C_VEL
LIN {X 0,Y 425.281,Z 774.681,A -85,B 0,C 180,E1 -9870.279,E2 -9870.279} C_VEL
LIN {X 0,Y 425.082,Z 776.637,A -85,B 0,C 180,E1 -9873.486,E2 -9873.486} C_VEL
LIN {X 0,Y 424.866,Z 778.791,A -85,B 0,C 180,E1 -9876.608,E2 -9876.608} C_VEL
LIN {X 0,Y 424.735,Z 781.099,A -85,B 0,C 180,E1 -9879.666,E2 -9879.666} C_VEL
LIN {X 0,Y 424.599,Z 783.833,A -85,B 0,C 180,E1 -9883.028,E2 -9883.028} C_VEL
LIN {X 0,Y 428.138,Z 796.464,A -85,B 0,C 180,E1 -9883.724,E2 -9883.724} C_VEL
LIN {X 0,Y 429.231,Z 802.595,A -85,B 0,C 180,E1 -9884.081,E2 -9884.081} C_VEL
LIN {X 0,Y 428.658,Z 814.619,A -85,B 0,C 180,E1 -9884.791,E2 -9884.791} C_VEL
LIN {X 0,Y 427.971,Z 826.868,A -85,B 0,C 180,E1 -9885.739,E2 -9885.739} C_VEL
LIN {X 0,Y 427.247,Z 837.836,A -85,B 0,C 180,E1 -9886.806,E2 -9886.806} C_VEL
LIN {X 0,Y 426.565,Z 846.755,A -85,B 0,C 180,E1 -9887.873,E2 -9887.873} C_VEL
LIN {X 0,Y 425.964,Z 856.38,A -85,B 0,C 180,E1 -9889.302,E2 -9889.302} C_VEL
LIN {X 0,Y 425.396,Z 864.152,A -85,B 0,C 180,E1 -9890.729,E2 -9890.729} C_VEL
LIN {X 0,Y 425.006,Z 869.421,A -85,B 0,C 180,E1 -9891.919,E2 -9891.919} C_VEL
LIN {X 0,Y 424.778,Z 874.551,A -85,B 0,C 180,E1 -9893.348,E2 -9893.348} C_VEL
LIN {X 0,Y 424.433,Z 878.524,A -85,B 0,C 180,E1 -9894.774,E2 -9894.774} C_VEL
LIN {X 0,Y 424.419,Z 881.42,A -85,B 0,C 180,E1 -9896.201,E2 -9896.201} C_VEL
LIN {X 0,Y 424.302,Z 882.811,A -85,B 0,C 180,E1 -9897.151,E2 -9897.151} C_VEL
LIN {X 0,Y 424.294,Z 883.771,A -85,B 0,C 180,E1 -9898.101,E2 -9898.101} C_VEL
LIN {X 0,Y 424.253,Z 884.344,A -85,B 0,C 180,E1 -9899.05,E2 -9899.05} C_VEL
LIN {X 0,Y 424.219,Z 884.525,A -85,B 0,C 180,E1 -9899.999,E2 -9899.999} C_VEL
LIN {X 0,Y 424.235,Z 884.265,A -85,B 0,C 180,E1 -9900.948,E2 -9900.948} C_VEL
LIN {X 0,Y 424.261,Z 883.605,A -85,B 0,C 180,E1 -9901.898,E2 -9901.898} C_VEL
LIN {X 0,Y 424.276,Z 882.556,A -85,B 0,C 180,E1 -9902.847,E2 -9902.847} C_VEL
LIN {X 0,Y 424.377,Z 881.09,A -85,B 0,C 180,E1 -9903.797,E2 -9903.797} C_VEL
LIN {X 0,Y 424.384,Z 878.061,A -85,B 0,C 180,E1 -9905.225,E2 -9905.225} C_VEL
LIN {X 0,Y 424.624,Z 873.639,A -85,B 0,C 180,E1 -9906.749,E2 -9906.749} C_VEL
LIN {X 0,Y 424.962,Z 867.67,A -85,B 0,C 180,E1 -9908.319,E2 -9908.319} C_VEL
LIN {X 0,Y 425.417,Z 860.822,A -85,B 0,C 180,E1 -9909.748,E2 -9909.748} C_VEL
LIN {X 0,Y 425.972,Z 852.306,A -85,B 0,C 180,E1 -9911.177,E2 -9911.177} C_VEL
LIN {X 0,Y 426.539,Z 843.557,A -85,B 0,C 180,E1 -9912.367,E2 -9912.367} C_VEL
LIN {X 0,Y 427.193,Z 833.737,A -85,B 0,C 180,E1 -9913.464,E2 -9913.464} C_VEL
LIN {X 0,Y 427.779,Z 822.207,A -85,B 0,C 180,E1 -9914.509,E2 -9914.509} C_VEL
LIN {X 0,Y 428.37,Z 810.526,A -85,B 0,C 180,E1 -9915.334,E2 -9915.334} C_VEL
LIN {X 0,Y 428.715,Z 801.486,A -85,B 0,C 180,E1 -9915.849,E2 -9915.849} C_VEL
LIN {X 0,Y 426.48,Z 790.207,A -85,B 0,C 180,E1 -9916.436,E2 -9916.436} C_VEL
LIN {X 0,Y 424.279,Z 780.971,A -85,B 0,C 180,E1 -9916.846,E2 -9916.846} C_VEL
LIN {X 0,Y 424.339,Z 777.357,A -85,B 0,C 180,E1 -9920.352,E2 -9920.352} C_VEL
LIN {X 0,Y 424.403,Z 774.26,A -85,B 0,C 180,E1 -9923.417,E2 -9923.417} C_VEL
LIN {X 0,Y 424.517,Z 771.069,A -85,B 0,C 180,E1 -9926.621,E2 -9926.621} C_VEL
LIN {X 0,Y 424.507,Z 769.052,A -85,B 0,C 180,E1 -9928.692,E2 -9928.692} C_VEL
LIN {X 0,Y 424.699,Z 768.586,A -85,B 0,C 180,E1 -9930.626,E2 -9930.626} C_VEL
LIN {X 0,Y 425.009,Z 768.544,A -85,B 0,C 180,E1 -9933.071,E2 -9933.071} C_VEL
LIN {X 0,Y 425.216,Z 768.518,A -85,B 0,C 180,E1 -9935.916,E2 -9935.916} C_VEL
LIN {X 0,Y 425.289,Z 768.511,A -85,B 0,C 180,E1 -9939.042,E2 -9939.042} C_VEL
LIN {X 0,Y 425.27,Z 768.511,A -85,B 0,C 180,E1 -9942.652,E2 -9942.652} C_VEL
LIN {X 0,Y 425.256,Z 768.512,A -85,B 0,C 180,E1 -9946.043,E2 -9946.043} C_VEL
LIN {X 0,Y 425.268,Z 768.511,A -85,B 0,C 180,E1 -9948.62,E2 -9948.62} C_VEL
LIN {X 0,Y 425.295,Z 768.51,A -85,B 0,C 180,E1 -9951.101,E2 -9951.101} C_VEL
LIN {X 0,Y 425.291,Z 768.507,A -85,B 0,C 180,E1 -9954.663,E2 -9954.663} C_VEL
LIN {X 0,Y 425.256,Z 768.511,A -85,B 0,C 180,E1 -9958.072,E2 -9958.072} C_VEL
LIN {X 0,Y 425.306,Z 768.51,A -85,B 0,C 180,E1 -9961.366,E2 -9961.366} C_VEL
LIN {X 0,Y 425.262,Z 768.51,A -85,B 0,C 180,E1 -9964.552,E2 -9964.552} C_VEL
LIN {X 0,Y 425.275,Z 768.508,A -85,B 0,C 180,E1 -9966.633,E2 -9966.633} C_VEL
LIN {X 0,Y 425.286,Z 768.511,A -85,B 0,C 180,E1 -9969.694,E2 -9969.694} C_VEL
LIN {X 0,Y 425.323,Z 768.502,A -85,B 0,C 180,E1 -9972.697,E2 -9972.697} C_VEL
LIN {X 0,Y 425.337,Z 768.506,A -85,B 0,C 180,E1 -9975.65,E2 -9975.65} C_VEL
LIN {X 0,Y 425.338,Z 768.5,A -85,B 0,C 180,E1 -9978.564,E2 -9978.564} C_VEL
LIN {X 0,Y 425.396,Z 768.495,A -85,B 0,C 180,E1 -9981.449,E2 -9981.449} C_VEL
LIN {X 0,Y 425.499,Z 768.481,A -85,B 0,C 180,E1 -9984.312,E2 -9984.312} C_VEL
LIN {X 0,Y 425.553,Z 768.478,A -85,B 0,C 180,E1 -9988.107,E2 -9988.107} C_VEL
LIN {X 0,Y 425.561,Z 768.478,A -85,B 0,C 180,E1 -9990,E2 -9990} C_VEL
LIN {X 0,Y 425.499,Z 768.479,A -85,B 0,C 180,E1 -9992.84,E2 -9992.84} C_VEL
LIN {X 0,Y 425.387,Z 768.492,A -85,B 0,C 180,E1 -9995.145,E2 -9995.145} C_VEL
LIN {X 0,Y 424.813,Z 768.57,A -85,B 0,C 180,E1 -9995.937,E2 -9995.937} C_VEL
LIN {X 0,Y 421.961,Z 768.919,A -85,B 0,C 180,E1 -9997.221,E2 -9997.221} C_VEL
LIN {X 0,Y 419.481,Z 769.235,A -85,B 0,C 180,E1 -9998.259,E2 -9998.259} C_VEL
LIN {X 0,Y 418.403,Z 769.363,A -85,B 0,C 180,E1 -9999.061,E2 -9999.061} C_VEL
LIN {X 0,Y 418.311,Z 769.374,A -85,B 0,C 180,E1 -9999.333,E2 -9999.333} C_VEL
LIN {X 0,Y 418.336,Z 769.372,A -85,B 0,C 180,E1 -10003,E2 -10003} C_VEL
LIN {X 0,Y 418.302,Z 769.379,A -85,B 0,C 180,E1 -10006.735,E2 -10006.735} C_VEL
LIN {X 0,Y 418.261,Z 769.382,A -85,B 0,C 180,E1 -10009.79,E2 -10009.79} C_VEL
LIN {X 0,Y 418.222,Z 769.39,A -85,B 0,C 180,E1 -10012.737,E2 -10012.737} C_VEL
LIN {X 0,Y 418.225,Z 769.386,A -85,B 0,C 180,E1 -10015.907,E2 -10015.907} C_VEL
LIN {X 0,Y 418.252,Z 769.384,A -85,B 0,C 180,E1 -10019.163,E2 -10019.163} C_VEL
LIN {X 0,Y 418.249,Z 769.388,A -85,B 0,C 180,E1 -10022.845,E2 -10022.845} C_VEL
LIN {X 0,Y 418.237,Z 769.386,A -85,B 0,C 180,E1 -10026.239,E2 -10026.239} C_VEL
LIN {X 0,Y 418.24,Z 769.385,A -85,B 0,C 180,E1 -10029.683,E2 -10029.683} C_VEL
LIN {X 0,Y 418.223,Z 769.388,A -85,B 0,C 180,E1 -10032.322,E2 -10032.322} C_VEL
LIN {X 0,Y 418.23,Z 769.39,A -85,B 0,C 180,E1 -10035.11,E2 -10035.11} C_VEL
LIN {X 0,Y 418.235,Z 769.386,A -85,B 0,C 180,E1 -10037.768,E2 -10037.768} C_VEL
LIN {X 0,Y 418.248,Z 769.385,A -85,B 0,C 180,E1 -10040.621,E2 -10040.621} C_VEL
LIN {X 0,Y 418.194,Z 769.392,A -85,B 0,C 180,E1 -10043.972,E2 -10043.972} C_VEL
LIN {X 0,Y 418.055,Z 769.41,A -85,B 0,C 180,E1 -10046.307,E2 -10046.307} C_VEL
LIN {X 0,Y 417.705,Z 769.455,A -85,B 0,C 180,E1 -10049.103,E2 -10049.103} C_VEL
LIN {X 0,Y 417.364,Z 769.5,A -85,B 0,C 180,E1 -10051.87,E2 -10051.87} C_VEL
LIN {X 0,Y 417.349,Z 770.477,A -85,B 0,C 180,E1 -10053.19,E2 -10053.19} C_VEL
LIN {X 0,Y 417.272,Z 773.669,A -85,B 0,C 180,E1 -10056.159,E2 -10056.159} C_VEL
LIN {X 0,Y 417.265,Z 777.02,A -85,B 0,C 180,E1 -10059.287,E2 -10059.287} C_VEL
LIN {X 0,Y 417.197,Z 780.884,A -85,B 0,C 180,E1 -10062.856,E2 -10062.856} C_VEL
LIN {X 0,Y 417.211,Z 781.077,A -85,B 0,C 180,E1 -10063.03,E2 -10063.03} C_VEL
LIN {X 0,Y 420.234,Z 794.013,A -85,B 0,C 180,E1 -10063.607,E2 -10063.607} C_VEL
LIN {X 0,Y 421.713,Z 801.731,A -85,B 0,C 180,E1 -10064.035,E2 -10064.035} C_VEL
LIN {X 0,Y 421.283,Z 813.975,A -85,B 0,C 180,E1 -10064.768,E2 -10064.768} C_VEL
LIN {X 0,Y 420.663,Z 825.088,A -85,B 0,C 180,E1 -10065.619,E2 -10065.619} C_VEL
LIN {X 0,Y 420.048,Z 836.282,A -85,B 0,C 180,E1 -10066.701,E2 -10066.701} C_VEL
LIN {X 0,Y 419.3,Z 846.429,A -85,B 0,C 180,E1 -10067.907,E2 -10067.907} C_VEL
LIN {X 0,Y 418.685,Z 856.171,A -85,B 0,C 180,E1 -10069.361,E2 -10069.361} C_VEL
LIN {X 0,Y 418.159,Z 864.032,A -85,B 0,C 180,E1 -10070.814,E2 -10070.814} C_VEL
LIN {X 0,Y 417.704,Z 870.303,A -85,B 0,C 180,E1 -10072.265,E2 -10072.265} C_VEL
LIN {X 0,Y 417.562,Z 874.772,A -85,B 0,C 180,E1 -10073.548,E2 -10073.548} C_VEL
LIN {X 0,Y 417.25,Z 879.127,A -85,B 0,C 180,E1 -10075.17,E2 -10075.17} C_VEL
LIN {X 0,Y 417.281,Z 881.106,A -85,B 0,C 180,E1 -10076.138,E2 -10076.138} C_VEL
LIN {X 0,Y 417.207,Z 882.669,A -85,B 0,C 180,E1 -10077.104,E2 -10077.104} C_VEL
LIN {X 0,Y 417.169,Z 883.766,A -85,B 0,C 180,E1 -10078.07,E2 -10078.07} C_VEL
LIN {X 0,Y 417.136,Z 884.471,A -85,B 0,C 180,E1 -10079.036,E2 -10079.036} C_VEL
LIN {X 0,Y 417.117,Z 884.788,A -85,B 0,C 180,E1 -10080.001,E2 -10080.001} C_VEL
LIN {X 0,Y 417.165,Z 884.669,A -85,B 0,C 180,E1 -10080.966,E2 -10080.966} C_VEL
LIN {X 0,Y 417.224,Z 883.21,A -85,B 0,C 180,E1 -10082.898,E2 -10082.898} C_VEL
LIN {X 0,Y 417.353,Z 881.871,A -85,B 0,C 180,E1 -10083.863,E2 -10083.863} C_VEL
LIN {X 0,Y 417.358,Z 879.037,A -85,B 0,C 180,E1 -10085.315,E2 -10085.315} C_VEL
LIN {X 0,Y 417.709,Z 874.606,A -85,B 0,C 180,E1 -10086.934,E2 -10086.934} C_VEL
LIN {X 0,Y 417.955,Z 870.102,A -85,B 0,C 180,E1 -10088.218,E2 -10088.218} C_VEL
LIN {X 0,Y 418.44,Z 863.732,A -85,B 0,C 180,E1 -10089.67,E2 -10089.67} C_VEL
LIN {X 0,Y 419.076,Z 855.825,A -85,B 0,C 180,E1 -10091.121,E2 -10091.121} C_VEL
LIN {X 0,Y 419.625,Z 847.75,A -85,B 0,C 180,E1 -10092.331,E2 -10092.331} C_VEL
LIN {X 0,Y 420.389,Z 837.828,A -85,B 0,C 180,E1 -10093.537,E2 -10093.537} C_VEL
LIN {X 0,Y 421.056,Z 826.883,A -85,B 0,C 180,E1 -10094.624,E2 -10094.624} C_VEL
LIN {X 0,Y 421.87,Z 814.536,A -85,B 0,C 180,E1 -10095.583,E2 -10095.583} C_VEL
LIN {X 0,Y 422.374,Z 802.742,A -85,B 0,C 180,E1 -10096.301,E2 -10096.301} C_VEL
LIN {X 0,Y 419.796,Z 791.292,A -85,B 0,C 180,E1 -10096.981,E2 -10096.981} C_VEL
LIN {X 0,Y 417.466,Z 783.569,A -85,B 0,C 180,E1 -10097.413,E2 -10097.413} C_VEL
LIN {X 0,Y 417.523,Z 781.146,A -85,B 0,C 180,E1 -10099.674,E2 -10099.674} C_VEL
LIN {X 0,Y 417.558,Z 777.825,A -85,B 0,C 180,E1 -10102.776,E2 -10102.776} C_VEL
LIN {X 0,Y 417.584,Z 774.298,A -85,B 0,C 180,E1 -10105.951,E2 -10105.951} C_VEL
LIN {X 0,Y 417.602,Z 770.57,A -85,B 0,C 180,E1 -10109.214,E2 -10109.214} C_VEL
LIN {X 0,Y 417.597,Z 769.471,A -85,B 0,C 180,E1 -10110.325,E2 -10110.325} C_VEL
LIN {X 0,Y 418.033,Z 769.416,A -85,B 0,C 180,E1 -10113.698,E2 -10113.698} C_VEL
LIN {X 0,Y 418.205,Z 769.391,A -85,B 0,C 180,E1 -10116.23,E2 -10116.23} C_VEL
LIN {X 0,Y 418.246,Z 769.387,A -85,B 0,C 180,E1 -10119.683,E2 -10119.683} C_VEL
LIN {X 0,Y 418.228,Z 769.388,A -85,B 0,C 180,E1 -10122.321,E2 -10122.321} C_VEL
LIN {X 0,Y 418.24,Z 769.39,A -85,B 0,C 180,E1 -10125.109,E2 -10125.109} C_VEL
LIN {X 0,Y 418.281,Z 769.459,A -85,B 0,C 180,E1 -10127.259,E2 -10127.259} C_VEL
LIN {X 0,Y 419.403,Z 775.697,A -85,B 0,C 180,E1 -10130.448,E2 -10130.448} C_VEL
LIN {X 0,Y 420.33,Z 781.742,A -85,B 0,C 180,E1 -10133.377,E2 -10133.377} C_VEL
LIN {X 0,Y 420.322,Z 785.326,A -85,B 0,C 180,E1 -10135.016,E2 -10135.016} C_VEL
LIN {X 0,Y 419.75,Z 792.495,A -85,B 0,C 180,E1 -10138.169,E2 -10138.169} C_VEL
LIN {X 0,Y 419.139,Z 800.21,A -85,B 0,C 180,E1 -10141.453,E2 -10141.453} C_VEL
LIN {X 0,Y 418.643,Z 807.896,A -85,B 0,C 180,E1 -10144.635,E2 -10144.635} C_VEL
LIN {X 0,Y 418.242,Z 815.09,A -85,B 0,C 180,E1 -10147.55,E2 -10147.55} C_VEL
LIN {X 0,Y 417.861,Z 823.4,A -85,B 0,C 180,E1 -10150.854,E2 -10150.854} C_VEL
LIN {X 0,Y 417.642,Z 828.451,A -85,B 0,C 180,E1 -10152.835,E2 -10152.835} C_VEL
LIN {X 0,Y 420.019,Z 844.672,A -85,B 0,C 180,E1 -10153.496,E2 -10153.496} C_VEL
LIN {X 0,Y 421.375,Z 856.75,A -85,B 0,C 180,E1 -10154.15,E2 -10154.15} C_VEL
LIN {X 0,Y 420.58,Z 869.556,A -85,B 0,C 180,E1 -10154.989,E2 -10154.989} C_VEL
LIN {X 0,Y 419.839,Z 881.422,A -85,B 0,C 180,E1 -10156,E2 -10156} C_VEL
LIN {X 0,Y 419.234,Z 891.277,A -85,B 0,C 180,E1 -10157.043,E2 -10157.043} C_VEL
LIN {X 0,Y 418.681,Z 899.793,A -85,B 0,C 180,E1 -10158.134,E2 -10158.134} C_VEL
LIN {X 0,Y 418.028,Z 909.047,A -85,B 0,C 180,E1 -10159.588,E2 -10159.588} C_VEL
LIN {X 0,Y 417.613,Z 916.502,A -85,B 0,C 180,E1 -10161.044,E2 -10161.044} C_VEL
LIN {X 0,Y 417.316,Z 923.352,A -85,B 0,C 180,E1 -10162.744,E2 -10162.744} C_VEL
LIN {X 0,Y 417.151,Z 927.851,A -85,B 0,C 180,E1 -10164.198,E2 -10164.198} C_VEL
LIN {X 0,Y 417.162,Z 930.221,A -85,B 0,C 180,E1 -10165.168,E2 -10165.168} C_VEL
LIN {X 0,Y 417.056,Z 932.139,A -85,B 0,C 180,E1 -10166.135,E2 -10166.135} C_VEL
LIN {X 0,Y 417.116,Z 933.61,A -85,B 0,C 180,E1 -10167.103,E2 -10167.103} C_VEL
LIN {X 0,Y 417.119,Z 934.624,A -85,B 0,C 180,E1 -10168.069,E2 -10168.069} C_VEL
LIN {X 0,Y 417.118,Z 935.234,A -85,B 0,C 180,E1 -10169.035,E2 -10169.035} C_VEL
LIN {X 0,Y 417.146,Z 935.44,A -85,B 0,C 180,E1 -10170,E2 -10170} C_VEL
LIN {X 0,Y 417.118,Z 935.199,A -85,B 0,C 180,E1 -10170.965,E2 -10170.965} C_VEL
LIN {X 0,Y 417.121,Z 934.534,A -85,B 0,C 180,E1 -10171.931,E2 -10171.931} C_VEL
LIN {X 0,Y 417.139,Z 933.463,A -85,B 0,C 180,E1 -10172.897,E2 -10172.897} C_VEL
LIN {X 0,Y 417.076,Z 931.968,A -85,B 0,C 180,E1 -10173.865,E2 -10173.865} C_VEL
LIN {X 0,Y 417.196,Z 928.86,A -85,B 0,C 180,E1 -10175.316,E2 -10175.316} C_VEL
LIN {X 0,Y 417.246,Z 924.665,A -85,B 0,C 180,E1 -10176.771,E2 -10176.771} C_VEL
LIN {X 0,Y 417.525,Z 918.239,A -85,B 0,C 180,E1 -10178.47,E2 -10178.47} C_VEL
LIN {X 0,Y 417.891,Z 911.256,A -85,B 0,C 180,E1 -10179.926,E2 -10179.926} C_VEL
LIN {X 0,Y 418.412,Z 902.668,A -85,B 0,C 180,E1 -10181.383,E2 -10181.383} C_VEL
LIN {X 0,Y 418.972,Z 893.881,A -85,B 0,C 180,E1 -10182.596,E2 -10182.596} C_VEL
LIN {X 0,Y 419.662,Z 883.67,A -85,B 0,C 180,E1 -10183.754,E2 -10183.754} C_VEL
LIN {X 0,Y 420.407,Z 872.706,A -85,B 0,C 180,E1 -10184.77,E2 -10184.77} C_VEL
LIN {X 0,Y 421.181,Z 861.397,A -85,B 0,C 180,E1 -10185.609,E2 -10185.609} C_VEL
LIN {X 0,Y 421.324,Z 854.527,A -85,B 0,C 180,E1 -10186.038,E2 -10186.038} C_VEL
LIN {X 0,Y 420.104,Z 842.725,A -85,B 0,C 180,E1 -10186.715,E2 -10186.715} C_VEL
LIN {X 0,Y 418.457,Z 830.527,A -85,B 0,C 180,E1 -10187.274,E2 -10187.274} C_VEL
LIN {X 0,Y 417.626,Z 825.727,A -85,B 0,C 180,E1 -10187.481,E2 -10187.481} C_VEL
LIN {X 0,Y 417.931,Z 816.118,A -85,B 0,C 180,E1 -10191.195,E2 -10191.195} C_VEL
LIN {X 0,Y 418.305,Z 808.403,A -85,B 0,C 180,E1 -10194.307,E2 -10194.307} C_VEL
LIN {X 0,Y 418.722,Z 801.633,A -85,B 0,C 180,E1 -10197.179,E2 -10197.179} C_VEL
LIN {X 0,Y 419.34,Z 793.86,A -85,B 0,C 180,E1 -10200.742,E2 -10200.742} C_VEL
LIN {X 0,Y 420.021,Z 788.369,A -85,B 0,C 180,E1 -10203.516,E2 -10203.516} C_VEL
LIN {X 0,Y 420.373,Z 784.355,A -85,B 0,C 180,E1 -10205.814,E2 -10205.814} C_VEL
LIN {X 0,Y 420.189,Z 780.804,A -85,B 0,C 180,E1 -10208.233,E2 -10208.233} C_VEL
LIN {X 0,Y 419.699,Z 777.483,A -85,B 0,C 180,E1 -10211.101,E2 -10211.101} C_VEL
LIN {X 0,Y 419.289,Z 775.168,A -85,B 0,C 180,E1 -10213.882,E2 -10213.882} C_VEL
LIN {X 0,Y 418.982,Z 773.765,A -85,B 0,C 180,E1 -10216.548,E2 -10216.548} C_VEL
LIN {X 0,Y 418.875,Z 773.079,A -85,B 0,C 180,E1 -10219.129,E2 -10219.129} C_VEL
LIN {X 0,Y 418.815,Z 773.027,A -85,B 0,C 180,E1 -10222.064,E2 -10222.064} C_VEL
LIN {X 0,Y 418.751,Z 773.672,A -85,B 0,C 180,E1 -10225.205,E2 -10225.205} C_VEL
LIN {X 0,Y 418.567,Z 774.518,A -85,B 0,C 180,E1 -10227.499,E2 -10227.499} C_VEL
LIN {X 0,Y 418.234,Z 776.208,A -85,B 0,C 180,E1 -10230.905,E2 -10230.905} C_VEL
LIN {X 0,Y 417.999,Z 778.117,A -85,B 0,C 180,E1 -10234.077,E2 -10234.077} C_VEL
LIN {X 0,Y 417.801,Z 780.281,A -85,B 0,C 180,E1 -10237.238,E2 -10237.238} C_VEL
LIN {X 0,Y 417.679,Z 782.672,A -85,B 0,C 180,E1 -10240.438,E2 -10240.438} C_VEL
LIN {X 0,Y 417.563,Z 784.549,A -85,B 0,C 180,E1 -10242.695,E2 -10242.695} C_VEL
LIN {X 0,Y 421.155,Z 796.688,A -85,B 0,C 180,E1 -10243.374,E2 -10243.374} C_VEL
LIN {X 0,Y 422.527,Z 803.483,A -85,B 0,C 180,E1 -10243.794,E2 -10243.794} C_VEL
LIN {X 0,Y 421.876,Z 815.67,A -85,B 0,C 180,E1 -10244.54,E2 -10244.54} C_VEL
LIN {X 0,Y 421.163,Z 827.702,A -85,B 0,C 180,E1 -10245.503,E2 -10245.503} C_VEL
LIN {X 0,Y 420.376,Z 838.577,A -85,B 0,C 180,E1 -10246.586,E2 -10246.586} C_VEL
LIN {X 0,Y 419.525,Z 849.182,A -85,B 0,C 180,E1 -10247.912,E2 -10247.912} C_VEL
LIN {X 0,Y 419.026,Z 857.038,A -85,B 0,C 180,E1 -10249.123,E2 -10249.123} C_VEL
LIN {X 0,Y 418.419,Z 864.77,A -85,B 0,C 180,E1 -10250.573,E2 -10250.573} C_VEL
LIN {X 0,Y 418.017,Z 869.997,A -85,B 0,C 180,E1 -10251.783,E2 -10251.783} C_VEL
LIN {X 0,Y 417.739,Z 875.086,A -85,B 0,C 180,E1 -10253.236,E2 -10253.236} C_VEL
LIN {X 0,Y 417.377,Z 879.029,A -85,B 0,C 180,E1 -10254.685,E2 -10254.685} C_VEL
LIN {X 0,Y 417.365,Z 881.912,A -85,B 0,C 180,E1 -10256.137,E2 -10256.137} C_VEL
LIN {X 0,Y 417.24,Z 883.289,A -85,B 0,C 180,E1 -10257.103,E2 -10257.103} C_VEL
LIN {X 0,Y 417.213,Z 884.24,A -85,B 0,C 180,E1 -10258.068,E2 -10258.068} C_VEL
LIN {X 0,Y 417.181,Z 884.8,A -85,B 0,C 180,E1 -10259.034,E2 -10259.034} C_VEL
LIN {X 0,Y 417.146,Z 884.966,A -85,B 0,C 180,E1 -10259.999,E2 -10259.999} C_VEL
LIN {X 0,Y 417.15,Z 884.689,A -85,B 0,C 180,E1 -10260.964,E2 -10260.964} C_VEL
LIN {X 0,Y 417.182,Z 884.013,A -85,B 0,C 180,E1 -10261.93,E2 -10261.93} C_VEL
LIN {X 0,Y 417.215,Z 882.943,A -85,B 0,C 180,E1 -10262.896,E2 -10262.896} C_VEL
LIN {X 0,Y 417.302,Z 881.452,A -85,B 0,C 180,E1 -10263.862,E2 -10263.862} C_VEL
LIN {X 0,Y 417.335,Z 878.388,A -85,B 0,C 180,E1 -10265.313,E2 -10265.313} C_VEL
LIN {X 0,Y 417.588,Z 873.598,A -85,B 0,C 180,E1 -10266.958,E2 -10266.958} C_VEL
LIN {X 0,Y 418.009,Z 866.876,A -85,B 0,C 180,E1 -10268.702,E2 -10268.702} C_VEL
LIN {X 0,Y 418.468,Z 859.704,A -85,B 0,C 180,E1 -10270.156,E2 -10270.156} C_VEL
LIN {X 0,Y 419.043,Z 850.774,A -85,B 0,C 180,E1 -10271.609,E2 -10271.609} C_VEL
LIN {X 0,Y 419.738,Z 841.645,A -85,B 0,C 180,E1 -10272.817,E2 -10272.817} C_VEL
LIN {X 0,Y 420.452,Z 830.577,A -85,B 0,C 180,E1 -10273.999,E2 -10273.999} C_VEL
LIN {X 0,Y 421.06,Z 818.955,A -85,B 0,C 180,E1 -10274.993,E2 -10274.993} C_VEL
LIN {X 0,Y 421.719,Z 806.971,A -85,B 0,C 180,E1 -10275.79,E2 -10275.79} C_VEL
LIN {X 0,Y 421.664,Z 801.097,A -85,B 0,C 180,E1 -10276.119,E2 -10276.119} C_VEL
LIN {X 0,Y 418.766,Z 787.929,A -85,B 0,C 180,E1 -10276.807,E2 -10276.807} C_VEL
LIN {X 0,Y 417.227,Z 781.313,A -85,B 0,C 180,E1 -10277.112,E2 -10277.112} C_VEL
LIN {X 0,Y 417.245,Z 778.667,A -85,B 0,C 180,E1 -10279.685,E2 -10279.685} C_VEL
LIN {X 0,Y 417.313,Z 775.542,A -85,B 0,C 180,E1 -10282.788,E2 -10282.788} C_VEL
LIN {X 0,Y 417.405,Z 772.394,A -85,B 0,C 180,E1 -10285.96,E2 -10285.96} C_VEL
LIN {X 0,Y 417.459,Z 769.534,A -85,B 0,C 180,E1 -10288.904,E2 -10288.904} C_VEL
LIN {X 0,Y 417.762,Z 769.447,A -85,B 0,C 180,E1 -10291.432,E2 -10291.432} C_VEL
LIN {X 0,Y 418.124,Z 769.404,A -85,B 0,C 180,E1 -10294.852,E2 -10294.852} C_VEL
LIN {X 0,Y 418.221,Z 769.389,A -85,B 0,C 180,E1 -10297.832,E2 -10297.832} C_VEL
LIN {X 0,Y 418.217,Z 769.393,A -85,B 0,C 180,E1 -10300.947,E2 -10300.947} C_VEL
LIN {X 0,Y 418.205,Z 769.39,A -85,B 0,C 180,E1 -10303.728,E2 -10303.728} C_VEL
LIN {X 0,Y 418.203,Z 769.391,A -85,B 0,C 180,E1 -10306.448,E2 -10306.448} C_VEL
LIN {X 0,Y 418.217,Z 769.393,A -85,B 0,C 180,E1 -10309.129,E2 -10309.129} C_VEL
LIN {X 0,Y 418.22,Z 769.388,A -85,B 0,C 180,E1 -10312.166,E2 -10312.166} C_VEL
LIN {X 0,Y 418.257,Z 769.386,A -85,B 0,C 180,E1 -10315.419,E2 -10315.419} C_VEL
LIN {X 0,Y 418.203,Z 769.39,A -85,B 0,C 180,E1 -10318.603,E2 -10318.603} C_VEL
LIN {X 0,Y 418.24,Z 769.386,A -85,B 0,C 180,E1 -10321.933,E2 -10321.933} C_VEL
LIN {X 0,Y 418.264,Z 769.384,A -85,B 0,C 180,E1 -10325.161,E2 -10325.161} C_VEL
LIN {X 0,Y 418.225,Z 769.386,A -85,B 0,C 180,E1 -10328.303,E2 -10328.303} C_VEL
LIN {X 0,Y 418.266,Z 769.384,A -85,B 0,C 180,E1 -10331.382,E2 -10331.382} C_VEL
LIN {X 0,Y 418.292,Z 769.378,A -85,B 0,C 180,E1 -10334.405,E2 -10334.405} C_VEL
LIN {X 0,Y 418.346,Z 769.373,A -85,B 0,C 180,E1 -10337.385,E2 -10337.385} C_VEL
LIN {X 0,Y 418.325,Z 769.374,A -85,B 0,C 180,E1 -10340.328,E2 -10340.328} C_VEL
LIN {X 0,Y 418.43,Z 769.361,A -85,B 0,C 180,E1 -10343.248,E2 -10343.248} C_VEL
LIN {X 0,Y 418.303,Z 769.376,A -85,B 0,C 180,E1 -10345.181,E2 -10345.181} C_VEL
LIN {X 0,Y 418.522,Z 769.354,A -85,B 0,C 180,E1 -10348.075,E2 -10348.075} C_VEL
LIN {X 0,Y 418.395,Z 769.363,A -85,B 0,C 180,E1 -10350.962,E2 -10350.962} C_VEL
LIN {X 0,Y 418.456,Z 769.356,A -85,B 0,C 180,E1 -10352.888,E2 -10352.888} C_VEL
LIN {X 0,Y 418.458,Z 769.359,A -85,B 0,C 180,E1 -10355.784,E2 -10355.784} C_VEL
LIN {X 0,Y 418.355,Z 769.37,A -85,B 0,C 180,E1 -10358.696,E2 -10358.696} C_VEL
LIN {X 0,Y 418.311,Z 769.374,A -85,B 0,C 180,E1 -10359.333,E2 -10359.333} C_VEL
LIN {X 0,Y 417.641,Z 769.464,A -85,B 0,C 180,E1 -10360.137,E2 -10360.137} C_VEL
LIN {X 0,Y 414.805,Z 769.811,A -85,B 0,C 180,E1 -10361.443,E2 -10361.443} C_VEL
LIN {X 0,Y 412.397,Z 770.116,A -85,B 0,C 180,E1 -10362.497,E2 -10362.497} C_VEL
LIN {X 0,Y 411.348,Z 770.242,A -85,B 0,C 180,E1 -10363.312,E2 -10363.312} C_VEL
LIN {X 0,Y 411.254,Z 770.254,A -85,B 0,C 180,E1 -10363.588,E2 -10363.588} C_VEL
LIN {X 0,Y 411.248,Z 770.256,A -85,B 0,C 180,E1 -10366.889,E2 -10366.889} C_VEL
LIN {X 0,Y 411.222,Z 770.26,A -85,B 0,C 180,E1 -10369.987,E2 -10369.987} C_VEL
LIN {X 0,Y 411.186,Z 770.264,A -85,B 0,C 180,E1 -10373.149,E2 -10373.149} C_VEL
LIN {X 0,Y 411.177,Z 770.267,A -85,B 0,C 180,E1 -10376.385,E2 -10376.385} C_VEL
LIN {X 0,Y 411.19,Z 770.263,A -85,B 0,C 180,E1 -10379.714,E2 -10379.714} C_VEL
LIN {X 0,Y 411.199,Z 770.264,A -85,B 0,C 180,E1 -10383.157,E2 -10383.157} C_VEL
LIN {X 0,Y 411.185,Z 770.266,A -85,B 0,C 180,E1 -10386.553,E2 -10386.553} C_VEL
LIN {X 0,Y 411.204,Z 770.262,A -85,B 0,C 180,E1 -10389.728,E2 -10389.728} C_VEL
LIN {X 0,Y 411.167,Z 770.27,A -85,B 0,C 180,E1 -10393.135,E2 -10393.135} C_VEL
LIN {X 0,Y 411.163,Z 770.268,A -85,B 0,C 180,E1 -10395.882,E2 -10395.882} C_VEL
LIN {X 0,Y 411.159,Z 770.269,A -85,B 0,C 180,E1 -10398.773,E2 -10398.773} C_VEL
LIN {X 0,Y 411.199,Z 770.263,A -85,B 0,C 180,E1 -10401.833,E2 -10401.833} C_VEL
LIN {X 0,Y 411.097,Z 770.278,A -85,B 0,C 180,E1 -10405.145,E2 -10405.145} C_VEL
LIN {X 0,Y 410.822,Z 770.313,A -85,B 0,C 180,E1 -10407.974,E2 -10407.974} C_VEL
LIN {X 0,Y 410.385,Z 770.369,A -85,B 0,C 180,E1 -10411.348,E2 -10411.348} C_VEL
LIN {X 0,Y 410.251,Z 770.386,A -85,B 0,C 180,E1 -10412.45,E2 -10412.45} C_VEL
LIN {X 0,Y 410.227,Z 773.819,A -85,B 0,C 180,E1 -10415.723,E2 -10415.723} C_VEL
LIN {X 0,Y 410.179,Z 777.246,A -85,B 0,C 180,E1 -10418.913,E2 -10418.913} C_VEL
LIN {X 0,Y 410.119,Z 780.604,A -85,B 0,C 180,E1 -10422.035,E2 -10422.035} C_VEL
LIN {X 0,Y 410.12,Z 781.402,A -85,B 0,C 180,E1 -10422.763,E2 -10422.763} C_VEL
LIN {X 0,Y 413.079,Z 794.169,A -85,B 0,C 180,E1 -10423.346,E2 -10423.346} C_VEL
LIN {X 0,Y 414.751,Z 802.384,A -85,B 0,C 180,E1 -10423.817,E2 -10423.817} C_VEL
LIN {X 0,Y 414.511,Z 811.896,A -85,B 0,C 180,E1 -10424.387,E2 -10424.387} C_VEL
LIN {X 0,Y 413.86,Z 823.419,A -85,B 0,C 180,E1 -10425.244,E2 -10425.244} C_VEL
LIN {X 0,Y 413.259,Z 833.977,A -85,B 0,C 180,E1 -10426.227,E2 -10426.227} C_VEL
LIN {X 0,Y 412.517,Z 844.576,A -85,B 0,C 180,E1 -10427.455,E2 -10427.455} C_VEL
LIN {X 0,Y 411.911,Z 853.266,A -85,B 0,C 180,E1 -10428.686,E2 -10428.686} C_VEL
LIN {X 0,Y 411.342,Z 861.766,A -85,B 0,C 180,E1 -10430.164,E2 -10430.164} C_VEL
LIN {X 0,Y 410.821,Z 868.575,A -85,B 0,C 180,E1 -10431.64,E2 -10431.64} C_VEL
LIN {X 0,Y 410.487,Z 874.399,A -85,B 0,C 180,E1 -10433.231,E2 -10433.231} C_VEL
LIN {X 0,Y 410.293,Z 878.281,A -85,B 0,C 180,E1 -10434.595,E2 -10434.595} C_VEL
LIN {X 0,Y 410.192,Z 881.456,A -85,B 0,C 180,E1 -10436.071,E2 -10436.071} C_VEL
LIN {X 0,Y 410.147,Z 883.04,A -85,B 0,C 180,E1 -10437.054,E2 -10437.054} C_VEL
LIN {X 0,Y 410.094,Z 884.16,A -85,B 0,C 180,E1 -10438.037,E2 -10438.037} C_VEL
LIN {X 0,Y 410.054,Z 884.88,A -85,B 0,C 180,E1 -10439.019,E2 -10439.019} C_VEL
LIN {X 0,Y 410.033,Z 885.209,A -85,B 0,C 180,E1 -10440.001,E2 -10440.001} C_VEL
LIN {X 0,Y 410.082,Z 885.114,A -85,B 0,C 180,E1 -10440.983,E2 -10440.983} C_VEL
LIN {X 0,Y 410.166,Z 883.685,A -85,B 0,C 180,E1 -10442.947,E2 -10442.947} C_VEL
LIN {X 0,Y 410.298,Z 882.369,A -85,B 0,C 180,E1 -10443.93,E2 -10443.93} C_VEL
LIN {X 0,Y 410.31,Z 879.57,A -85,B 0,C 180,E1 -10445.407,E2 -10445.407} C_VEL
LIN {X 0,Y 410.67,Z 875.394,A -85,B 0,C 180,E1 -10446.981,E2 -10446.981} C_VEL
LIN {X 0,Y 410.951,Z 870.683,A -85,B 0,C 180,E1 -10448.359,E2 -10448.359} C_VEL
LIN {X 0,Y 411.47,Z 864.333,A -85,B 0,C 180,E1 -10449.835,E2 -10449.835} C_VEL
LIN {X 0,Y 412.148,Z 856.45,A -85,B 0,C 180,E1 -10451.31,E2 -10451.31} C_VEL
LIN {X 0,Y 412.725,Z 848.464,A -85,B 0,C 180,E1 -10452.54,E2 -10452.54} C_VEL
LIN {X 0,Y 413.542,Z 838.666,A -85,B 0,C 180,E1 -10453.765,E2 -10453.765} C_VEL
LIN {X 0,Y 414.258,Z 827.847,A -85,B 0,C 180,E1 -10454.869,E2 -10454.869} C_VEL
LIN {X 0,Y 415.03,Z 817.409,A -85,B 0,C 180,E1 -10455.721,E2 -10455.721} C_VEL
LIN {X 0,Y 415.706,Z 804.445,A -85,B 0,C 180,E1 -10456.548,E2 -10456.548} C_VEL
LIN {X 0,Y 413.121,Z 792.879,A -85,B 0,C 180,E1 -10457.282,E2 -10457.282} C_VEL
LIN {X 0,Y 410.431,Z 784.136,A -85,B 0,C 180,E1 -10457.79,E2 -10457.79} C_VEL
LIN {X 0,Y 410.482,Z 781.764,A -85,B 0,C 180,E1 -10460.026,E2 -10460.026} C_VEL
LIN {X 0,Y 410.532,Z 778.39,A -85,B 0,C 180,E1 -10463.188,E2 -10463.188} C_VEL
LIN {X 0,Y 410.563,Z 774.842,A -85,B 0,C 180,E1 -10466.429,E2 -10466.429} C_VEL
LIN {X 0,Y 410.571,Z 771.101,A -85,B 0,C 180,E1 -10469.764,E2 -10469.764} C_VEL
LIN {X 0,Y 410.683,Z 770.332,A -85,B 0,C 180,E1 -10471.168,E2 -10471.168} C_VEL
LIN {X 0,Y 411.042,Z 770.287,A -85,B 0,C 180,E1 -10474.35,E2 -10474.35} C_VEL
LIN {X 0,Y 411.176,Z 770.27,A -85,B 0,C 180,E1 -10476.744,E2 -10476.744} C_VEL
LIN {X 0,Y 411.211,Z 770.264,A -85,B 0,C 180,E1 -10479.727,E2 -10479.727} C_VEL
LIN {X 0,Y 411.175,Z 770.269,A -85,B 0,C 180,E1 -10483.134,E2 -10483.134} C_VEL
LIN {X 0,Y 411.217,Z 770.262,A -85,B 0,C 180,E1 -10486.934,E2 -10486.934} C_VEL
LIN {X 0,Y 412.305,Z 776.312,A -85,B 0,C 180,E1 -10490.091,E2 -10490.091} C_VEL
LIN {X 0,Y 413.301,Z 782.296,A -85,B 0,C 180,E1 -10493.056,E2 -10493.056} C_VEL
LIN {X 0,Y 413.351,Z 785.792,A -85,B 0,C 180,E1 -10494.699,E2 -10494.699} C_VEL
LIN {X 0,Y 412.837,Z 792.177,A -85,B 0,C 180,E1 -10497.571,E2 -10497.571} C_VEL
LIN {X 0,Y 412.29,Z 798.623,A -85,B 0,C 180,E1 -10500.385,E2 -10500.385} C_VEL
LIN {X 0,Y 411.665,Z 807.591,A -85,B 0,C 180,E1 -10504.193,E2 -10504.193} C_VEL
LIN {X 0,Y 411.193,Z 815.244,A -85,B 0,C 180,E1 -10507.363,E2 -10507.363} C_VEL
LIN {X 0,Y 410.803,Z 823.232,A -85,B 0,C 180,E1 -10510.607,E2 -10510.607} C_VEL
LIN {X 0,Y 410.592,Z 828.123,A -85,B 0,C 180,E1 -10512.57,E2 -10512.57} C_VEL
LIN {X 0,Y 412.915,Z 843.917,A -85,B 0,C 180,E1 -10513.226,E2 -10513.226} C_VEL
LIN {X 0,Y 414.382,Z 856.236,A -85,B 0,C 180,E1 -10513.909,E2 -10513.909} C_VEL
LIN {X 0,Y 413.679,Z 868.653,A -85,B 0,C 180,E1 -10514.732,E2 -10514.732} C_VEL
LIN {X 0,Y 412.881,Z 880.606,A -85,B 0,C 180,E1 -10515.761,E2 -10515.761} C_VEL
LIN {X 0,Y 412.198,Z 891.568,A -85,B 0,C 180,E1 -10516.943,E2 -10516.943} C_VEL
LIN {X 0,Y 411.559,Z 900.782,A -85,B 0,C 180,E1 -10518.175,E2 -10518.175} C_VEL
LIN {X 0,Y 410.93,Z 909.775,A -85,B 0,C 180,E1 -10519.655,E2 -10519.655} C_VEL
LIN {X 0,Y 410.518,Z 917.029,A -85,B 0,C 180,E1 -10521.137,E2 -10521.137} C_VEL
LIN {X 0,Y 410.258,Z 922.807,A -85,B 0,C 180,E1 -10522.618,E2 -10522.618} C_VEL
LIN {X 0,Y 410.078,Z 927.336,A -85,B 0,C 180,E1 -10524.098,E2 -10524.098} C_VEL
LIN {X 0,Y 410.095,Z 929.72,A -85,B 0,C 180,E1 -10525.084,E2 -10525.084} C_VEL
LIN {X 0,Y 409.973,Z 931.65,A -85,B 0,C 180,E1 -10526.068,E2 -10526.068} C_VEL
LIN {X 0,Y 410.018,Z 933.143,A -85,B 0,C 180,E1 -10527.052,E2 -10527.052} C_VEL
LIN {X 0,Y 410.046,Z 934.169,A -85,B 0,C 180,E1 -10528.036,E2 -10528.036} C_VEL
LIN {X 0,Y 410.036,Z 934.785,A -85,B 0,C 180,E1 -10529.018,E2 -10529.018} C_VEL
LIN {X 0,Y 410.061,Z 934.998,A -85,B 0,C 180,E1 -10530,E2 -10530} C_VEL
LIN {X 0,Y 410.037,Z 934.771,A -85,B 0,C 180,E1 -10530.982,E2 -10530.982} C_VEL
LIN {X 0,Y 410.048,Z 934.109,A -85,B 0,C 180,E1 -10531.964,E2 -10531.964} C_VEL
LIN {X 0,Y 410.04,Z 933.035,A -85,B 0,C 180,E1 -10532.947,E2 -10532.947} C_VEL
LIN {X 0,Y 409.991,Z 931.543,A -85,B 0,C 180,E1 -10533.932,E2 -10533.932} C_VEL
LIN {X 0,Y 410.111,Z 928.434,A -85,B 0,C 180,E1 -10535.408,E2 -10535.408} C_VEL
LIN {X 0,Y 410.179,Z 924.251,A -85,B 0,C 180,E1 -10536.889,E2 -10536.889} C_VEL
LIN {X 0,Y 410.481,Z 917.852,A -85,B 0,C 180,E1 -10538.616,E2 -10538.616} C_VEL
LIN {X 0,Y 410.854,Z 910.902,A -85,B 0,C 180,E1 -10540.098,E2 -10540.098} C_VEL
LIN {X 0,Y 411.415,Z 902.335,A -85,B 0,C 180,E1 -10541.579,E2 -10541.579} C_VEL
LIN {X 0,Y 412.011,Z 893.581,A -85,B 0,C 180,E1 -10542.812,E2 -10542.812} C_VEL
LIN {X 0,Y 412.76,Z 883.156,A -85,B 0,C 180,E1 -10544.017,E2 -10544.017} C_VEL
LIN {X 0,Y 413.652,Z 871.174,A -85,B 0,C 180,E1 -10545.143,E2 -10545.143} C_VEL
LIN {X 0,Y 414.608,Z 857.785,A -85,B 0,C 180,E1 -10546.115,E2 -10546.115} C_VEL
LIN {X 0,Y 413.514,Z 845.752,A -85,B 0,C 180,E1 -10546.873,E2 -10546.873} C_VEL
LIN {X 0,Y 412.031,Z 833.25,A -85,B 0,C 180,E1 -10547.497,E2 -10547.497} C_VEL
LIN {X 0,Y 410.59,Z 825.136,A -85,B 0,C 180,E1 -10547.877,E2 -10547.877} C_VEL
LIN {X 0,Y 410.919,Z 815.822,A -85,B 0,C 180,E1 -10551.575,E2 -10551.575} C_VEL
LIN {X 0,Y 411.387,Z 806.934,A -85,B 0,C 180,E1 -10555.283,E2 -10555.283} C_VEL
LIN {X 0,Y 411.877,Z 799.634,A -85,B 0,C 180,E1 -10558.54,E2 -10558.54} C_VEL
LIN {X 0,Y 412.601,Z 792.782,A -85,B 0,C 180,E1 -10561.873,E2 -10561.873} C_VEL
LIN {X 0,Y 413.168,Z 788.551,A -85,B 0,C 180,E1 -10564.148,E2 -10564.148} C_VEL
LIN {X 0,Y 413.423,Z 784.675,A -85,B 0,C 180,E1 -10566.512,E2 -10566.512} C_VEL
LIN {X 0,Y 413.107,Z 781.312,A -85,B 0,C 180,E1 -10569.011,E2 -10569.011} C_VEL
LIN {X 0,Y 412.686,Z 778.536,A -85,B 0,C 180,E1 -10571.619,E2 -10571.619} C_VEL
LIN {X 0,Y 412.315,Z 776.434,A -85,B 0,C 180,E1 -10574.335,E2 -10574.335} C_VEL
LIN {X 0,Y 412.017,Z 775.074,A -85,B 0,C 180,E1 -10577.179,E2 -10577.179} C_VEL
LIN {X 0,Y 411.906,Z 774.458,A -85,B 0,C 180,E1 -10580.157,E2 -10580.157} C_VEL
LIN {X 0,Y 411.825,Z 774.604,A -85,B 0,C 180,E1 -10583.329,E2 -10583.329} C_VEL
LIN {X 0,Y 411.74,Z 775.162,A -85,B 0,C 180,E1 -10585.716,E2 -10585.716} C_VEL
LIN {X 0,Y 411.385,Z 776.527,A -85,B 0,C 180,E1 -10589.168,E2 -10589.168} C_VEL
LIN {X 0,Y 411.108,Z 778.283,A -85,B 0,C 180,E1 -10592.51,E2 -10592.51} C_VEL
LIN {X 0,Y 410.873,Z 780.317,A -85,B 0,C 180,E1 -10595.762,E2 -10595.762} C_VEL
LIN {X 0,Y 410.728,Z 782.531,A -85,B 0,C 180,E1 -10598.94,E2 -10598.94} C_VEL
LIN {X 0,Y 410.537,Z 785.085,A -85,B 0,C 180,E1 -10602.277,E2 -10602.277} C_VEL
LIN {X 0,Y 414.551,Z 798.512,A -85,B 0,C 180,E1 -10603.109,E2 -10603.109} C_VEL
LIN {X 0,Y 415.795,Z 805.33,A -85,B 0,C 180,E1 -10603.546,E2 -10603.546} C_VEL
LIN {X 0,Y 414.994,Z 818.485,A -85,B 0,C 180,E1 -10604.404,E2 -10604.404} C_VEL
LIN {X 0,Y 414.255,Z 830.166,A -85,B 0,C 180,E1 -10605.39,E2 -10605.39} C_VEL
LIN {X 0,Y 413.347,Z 841.511,A -85,B 0,C 180,E1 -10606.604,E2 -10606.604} C_VEL
LIN {X 0,Y 412.622,Z 849.925,A -85,B 0,C 180,E1 -10607.706,E2 -10607.706} C_VEL
LIN {X 0,Y 411.968,Z 859.11,A -85,B 0,C 180,E1 -10609.183,E2 -10609.183} C_VEL
LIN {X 0,Y 411.36,Z 866.488,A -85,B 0,C 180,E1 -10610.658,E2 -10610.658} C_VEL
LIN {X 0,Y 410.852,Z 872.412,A -85,B 0,C 180,E1 -10612.134,E2 -10612.134} C_VEL
LIN {X 0,Y 410.61,Z 877.07,A -85,B 0,C 180,E1 -10613.611,E2 -10613.611} C_VEL
LIN {X 0,Y 410.283,Z 880.626,A -85,B 0,C 180,E1 -10615.086,E2 -10615.086} C_VEL
LIN {X 0,Y 410.311,Z 882.432,A -85,B 0,C 180,E1 -10616.07,E2 -10616.07} C_VEL
LIN {X 0,Y 410.181,Z 883.782,A -85,B 0,C 180,E1 -10617.053,E2 -10617.053} C_VEL
LIN {X 0,Y 410.136,Z 884.717,A -85,B 0,C 180,E1 -10618.035,E2 -10618.035} C_VEL
LIN {X 0,Y 410.097,Z 885.262,A -85,B 0,C 180,E1 -10619.017,E2 -10619.017} C_VEL
LIN {X 0,Y 410.061,Z 885.407,A -85,B 0,C 180,E1 -10619.999,E2 -10619.999} C_VEL
LIN {X 0,Y 410.067,Z 885.109,A -85,B 0,C 180,E1 -10620.981,E2 -10620.981} C_VEL
LIN {X 0,Y 410.107,Z 884.416,A -85,B 0,C 180,E1 -10621.963,E2 -10621.963} C_VEL
LIN {X 0,Y 410.155,Z 883.33,A -85,B 0,C 180,E1 -10622.946,E2 -10622.946} C_VEL
LIN {X 0,Y 410.213,Z 881.813,A -85,B 0,C 180,E1 -10623.929,E2 -10623.929} C_VEL
LIN {X 0,Y 410.29,Z 878.711,A -85,B 0,C 180,E1 -10625.405,E2 -10625.405} C_VEL
LIN {X 0,Y 410.514,Z 874.21,A -85,B 0,C 180,E1 -10626.979,E2 -10626.979} C_VEL
LIN {X 0,Y 410.899,Z 868.136,A -85,B 0,C 180,E1 -10628.606,E2 -10628.606} C_VEL
LIN {X 0,Y 411.371,Z 861.186,A -85,B 0,C 180,E1 -10630.084,E2 -10630.084} C_VEL
LIN {X 0,Y 411.987,Z 852.515,A -85,B 0,C 180,E1 -10631.562,E2 -10631.562} C_VEL
LIN {X 0,Y 412.642,Z 843.64,A -85,B 0,C 180,E1 -10632.791,E2 -10632.791} C_VEL
LIN {X 0,Y 413.359,Z 833.28,A -85,B 0,C 180,E1 -10633.967,E2 -10633.967} C_VEL
LIN {X 0,Y 414.015,Z 821.899,A -85,B 0,C 180,E1 -10635.002,E2 -10635.002} C_VEL
LIN {X 0,Y 414.682,Z 810.332,A -85,B 0,C 180,E1 -10635.832,E2 -10635.832} C_VEL
LIN {X 0,Y 414.978,Z 803.79,A -85,B 0,C 180,E1 -10636.221,E2 -10636.221} C_VEL
LIN {X 0,Y 412.618,Z 792.044,A -85,B 0,C 180,E1 -10636.885,E2 -10636.885} C_VEL
LIN {X 0,Y 410.133,Z 781.688,A -85,B 0,C 180,E1 -10637.352,E2 -10637.352} C_VEL
LIN {X 0,Y 410.17,Z 778.947,A -85,B 0,C 180,E1 -10640.039,E2 -10640.039} C_VEL
LIN {X 0,Y 410.255,Z 775.779,A -85,B 0,C 180,E1 -10643.203,E2 -10643.203} C_VEL
LIN {X 0,Y 410.356,Z 772.595,A -85,B 0,C 180,E1 -10646.441,E2 -10646.441} C_VEL
LIN {X 0,Y 410.388,Z 770.463,A -85,B 0,C 180,E1 -10648.652,E2 -10648.652} C_VEL
LIN {X 0,Y 410.784,Z 770.319,A -85,B 0,C 180,E1 -10652.029,E2 -10652.029} C_VEL
LIN {X 0,Y 411.085,Z 770.28,A -85,B 0,C 180,E1 -10654.853,E2 -10654.853} C_VEL
LIN {X 0,Y 411.198,Z 770.264,A -85,B 0,C 180,E1 -10658.167,E2 -10658.167} C_VEL
LIN {X 0,Y 411.159,Z 770.269,A -85,B 0,C 180,E1 -10661.227,E2 -10661.227} C_VEL
LIN {X 0,Y 411.171,Z 770.267,A -85,B 0,C 180,E1 -10664.489,E2 -10664.489} C_VEL
LIN {X 0,Y 411.171,Z 770.267,A -85,B 0,C 180,E1 -10668.194,E2 -10668.194} C_VEL
LIN {X 0,Y 411.208,Z 770.263,A -85,B 0,C 180,E1 -10670.774,E2 -10670.774} C_VEL
LIN {X 0,Y 411.19,Z 770.264,A -85,B 0,C 180,E1 -10674.47,E2 -10674.47} C_VEL
LIN {X 0,Y 411.2,Z 770.264,A -85,B 0,C 180,E1 -10676.873,E2 -10676.873} C_VEL
LIN {X 0,Y 411.204,Z 770.262,A -85,B 0,C 180,E1 -10680.649,E2 -10680.649} C_VEL
LIN {X 0,Y 411.186,Z 770.267,A -85,B 0,C 180,E1 -10683.615,E2 -10683.615} C_VEL
LIN {X 0,Y 411.186,Z 770.264,A -85,B 0,C 180,E1 -10686.851,E2 -10686.851} C_VEL
LIN {X 0,Y 411.205,Z 770.262,A -85,B 0,C 180,E1 -10690.05,E2 -10690.05} C_VEL
LIN {X 0,Y 411.254,Z 770.256,A -85,B 0,C 180,E1 -10693.131,E2 -10693.131} C_VEL
LIN {X 0,Y 411.296,Z 770.249,A -85,B 0,C 180,E1 -10696.896,E2 -10696.896} C_VEL
LIN {X 0,Y 411.277,Z 770.253,A -85,B 0,C 180,E1 -10700.161,E2 -10700.161} C_VEL
LIN {X 0,Y 411.38,Z 770.238,A -85,B 0,C 180,E1 -10703.132,E2 -10703.132} C_VEL
LIN {X 0,Y 411.275,Z 770.251,A -85,B 0,C 180,E1 -10705.099,E2 -10705.099} C_VEL
LIN {X 0,Y 411.491,Z 770.23,A -85,B 0,C 180,E1 -10708.042,E2 -10708.042} C_VEL
LIN {X 0,Y 411.365,Z 770.239,A -85,B 0,C 180,E1 -10710.979,E2 -10710.979} C_VEL
LIN {X 0,Y 411.414,Z 770.233,A -85,B 0,C 180,E1 -10712.938,E2 -10712.938} C_VEL
LIN {X 0,Y 411.379,Z 770.238,A -85,B 0,C 180,E1 -10716.868,E2 -10716.868} C_VEL
LIN {X 0,Y 411.264,Z 770.255,A -85,B 0,C 180,E1 -10719.839,E2 -10719.839} C_VEL
LIN {X 0,Y 411.295,Z 770.249,A -85,B 0,C 180,E1 -10723.104,E2 -10723.104} C_VEL
LIN {X 0,Y 411.254,Z 770.254,A -85,B 0,C 180,E1 -10723.588,E2 -10723.588} C_VEL
LIN {X 0,Y 410.558,Z 770.347,A -85,B 0,C 180,E1 -10724.406,E2 -10724.406} C_VEL
LIN {X 0,Y 407.68,Z 770.7,A -85,B 0,C 180,E1 -10725.734,E2 -10725.734} C_VEL
LIN {X 0,Y 405.271,Z 771.001,A -85,B 0,C 180,E1 -10726.807,E2 -10726.807} C_VEL
LIN {X 0,Y 404.254,Z 771.126,A -85,B 0,C 180,E1 -10727.636,E2 -10727.636} C_VEL
LIN {X 0,Y 404.179,Z 771.136,A -85,B 0,C 180,E1 -10727.917,E2 -10727.917} C_VEL
LIN {X 0,Y 404.155,Z 771.143,A -85,B 0,C 180,E1 -10730.352,E2 -10730.352} C_VEL
LIN {X 0,Y 404.148,Z 771.139,A -85,B 0,C 180,E1 -10733.576,E2 -10733.576} C_VEL
LIN {X 0,Y 404.122,Z 771.146,A -85,B 0,C 180,E1 -10736.883,E2 -10736.883} C_VEL
LIN {X 0,Y 404.136,Z 771.143,A -85,B 0,C 180,E1 -10740.286,E2 -10740.286} C_VEL
LIN {X 0,Y 404.137,Z 771.141,A -85,B 0,C 180,E1 -10743.813,E2 -10743.813} C_VEL
LIN {X 0,Y 404.129,Z 771.148,A -85,B 0,C 180,E1 -10746.876,E2 -10746.876} C_VEL
LIN {X 0,Y 404.141,Z 771.141,A -85,B 0,C 180,E1 -10750.081,E2 -10750.081} C_VEL
LIN {X 0,Y 404.147,Z 771.145,A -85,B 0,C 180,E1 -10753.085,E2 -10753.085} C_VEL
LIN {X 0,Y 404.143,Z 771.142,A -85,B 0,C 180,E1 -10755.927,E2 -10755.927} C_VEL
LIN {X 0,Y 404.113,Z 771.146,A -85,B 0,C 180,E1 -10758.636,E2 -10758.636} C_VEL
LIN {X 0,Y 404.148,Z 771.143,A -85,B 0,C 180,E1 -10761.494,E2 -10761.494} C_VEL
LIN {X 0,Y 404.063,Z 771.153,A -85,B 0,C 180,E1 -10764.973,E2 -10764.973} C_VEL
LIN {X 0,Y 403.847,Z 771.183,A -85,B 0,C 180,E1 -10767.353,E2 -10767.353} C_VEL
LIN {X 0,Y 403.414,Z 771.235,A -85,B 0,C 180,E1 -10770.806,E2 -10770.806} C_VEL
LIN {X 0,Y 403.2,Z 771.286,A -85,B 0,C 180,E1 -10772.743,E2 -10772.743} C_VEL
LIN {X 0,Y 403.118,Z 775.13,A -85,B 0,C 180,E1 -10776.362,E2 -10776.362} C_VEL
LIN {X 0,Y 403.085,Z 778.591,A -85,B 0,C 180,E1 -10779.593,E2 -10779.593} C_VEL
LIN {X 0,Y 403.081,Z 781.745,A -85,B 0,C 180,E1 -10782.506,E2 -10782.506} C_VEL
LIN {X 0,Y 406.11,Z 795.112,A -85,B 0,C 180,E1 -10783.13,E2 -10783.13} C_VEL
LIN {X 0,Y 407.968,Z 804.343,A -85,B 0,C 180,E1 -10783.677,E2 -10783.677} C_VEL
LIN {X 0,Y 407.348,Z 816.885,A -85,B 0,C 180,E1 -10784.49,E2 -10784.49} C_VEL
LIN {X 0,Y 406.622,Z 829.058,A -85,B 0,C 180,E1 -10785.512,E2 -10785.512} C_VEL
LIN {X 0,Y 405.977,Z 839.499,A -85,B 0,C 180,E1 -10786.613,E2 -10786.613} C_VEL
LIN {X 0,Y 405.121,Z 850.018,A -85,B 0,C 180,E1 -10787.986,E2 -10787.986} C_VEL
LIN {X 0,Y 404.594,Z 857.851,A -85,B 0,C 180,E1 -10789.239,E2 -10789.239} C_VEL
LIN {X 0,Y 404.043,Z 865.516,A -85,B 0,C 180,E1 -10790.742,E2 -10790.742} C_VEL
LIN {X 0,Y 403.544,Z 872.583,A -85,B 0,C 180,E1 -10792.496,E2 -10792.496} C_VEL
LIN {X 0,Y 403.361,Z 877.276,A -85,B 0,C 180,E1 -10794,E2 -10794} C_VEL
LIN {X 0,Y 403.09,Z 880.849,A -85,B 0,C 180,E1 -10795.501,E2 -10795.501} C_VEL
LIN {X 0,Y 403.087,Z 883.39,A -85,B 0,C 180,E1 -10797.003,E2 -10797.003} C_VEL
LIN {X 0,Y 403.023,Z 884.543,A -85,B 0,C 180,E1 -10798.002,E2 -10798.002} C_VEL
LIN {X 0,Y 402.953,Z 885.634,A -85,B 0,C 180,E1 -10800.001,E2 -10800.001} C_VEL
LIN {X 0,Y 403.002,Z 885.571,A -85,B 0,C 180,E1 -10801,E2 -10801} C_VEL
LIN {X 0,Y 403.109,Z 884.173,A -85,B 0,C 180,E1 -10802.999,E2 -10802.999} C_VEL
LIN {X 0,Y 403.244,Z 882.877,A -85,B 0,C 180,E1 -10803.999,E2 -10803.999} C_VEL
LIN {X 0,Y 403.267,Z 880.102,A -85,B 0,C 180,E1 -10805.501,E2 -10805.501} C_VEL
LIN {X 0,Y 403.652,Z 876.111,A -85,B 0,C 180,E1 -10807.052,E2 -10807.052} C_VEL
LIN {X 0,Y 403.962,Z 871.284,A -85,B 0,C 180,E1 -10808.505,E2 -10808.505} C_VEL
LIN {X 0,Y 404.509,Z 864.999,A -85,B 0,C 180,E1 -10810.006,E2 -10810.006} C_VEL
LIN {X 0,Y 405.228,Z 857.197,A -85,B 0,C 180,E1 -10811.506,E2 -10811.506} C_VEL
LIN {X 0,Y 405.839,Z 849.262,A -85,B 0,C 180,E1 -10812.757,E2 -10812.757} C_VEL
LIN {X 0,Y 406.704,Z 839.547,A -85,B 0,C 180,E1 -10814.001,E2 -10814.001} C_VEL
LIN {X 0,Y 407.471,Z 828.819,A -85,B 0,C 180,E1 -10815.123,E2 -10815.123} C_VEL
LIN {X 0,Y 408.395,Z 816.999,A -85,B 0,C 180,E1 -10816.106,E2 -10816.106} C_VEL
LIN {X 0,Y 409.051,Z 805.823,A -85,B 0,C 180,E1 -10816.838,E2 -10816.838} C_VEL
LIN {X 0,Y 406.493,Z 794.503,A -85,B 0,C 180,E1 -10817.596,E2 -10817.596} C_VEL
LIN {X 0,Y 403.428,Z 784.714,A -85,B 0,C 180,E1 -10818.193,E2 -10818.193} C_VEL
LIN {X 0,Y 403.428,Z 782.397,A -85,B 0,C 180,E1 -10820.391,E2 -10820.391} C_VEL
LIN {X 0,Y 403.503,Z 778.983,A -85,B 0,C 180,E1 -10823.617,E2 -10823.617} C_VEL
LIN {X 0,Y 403.562,Z 775.378,A -85,B 0,C 180,E1 -10826.924,E2 -10826.924} C_VEL
LIN {X 0,Y 403.576,Z 771.674,A -85,B 0,C 180,E1 -10830.333,E2 -10830.333} C_VEL
LIN {X 0,Y 403.667,Z 771.206,A -85,B 0,C 180,E1 -10831.488,E2 -10831.488} C_VEL
LIN {X 0,Y 403.946,Z 771.171,A -85,B 0,C 180,E1 -10833.832,E2 -10833.832} C_VEL
LIN {X 0,Y 404.124,Z 771.148,A -85,B 0,C 180,E1 -10836.872,E2 -10836.872} C_VEL
LIN {X 0,Y 404.152,Z 771.143,A -85,B 0,C 180,E1 -10840.08,E2 -10840.08} C_VEL
LIN {X 0,Y 404.155,Z 771.144,A -85,B 0,C 180,E1 -10843.084,E2 -10843.084} C_VEL
LIN {X 0,Y 404.178,Z 771.25,A -85,B 0,C 180,E1 -10846.71,E2 -10846.71} C_VEL
LIN {X 0,Y 405.219,Z 776.942,A -85,B 0,C 180,E1 -10849.741,E2 -10849.741} C_VEL
LIN {X 0,Y 406.213,Z 782.845,A -85,B 0,C 180,E1 -10852.738,E2 -10852.738} C_VEL
LIN {X 0,Y 406.396,Z 786.232,A -85,B 0,C 180,E1 -10854.371,E2 -10854.371} C_VEL
LIN {X 0,Y 405.823,Z 793.123,A -85,B 0,C 180,E1 -10857.53,E2 -10857.53} C_VEL
LIN {X 0,Y 405.307,Z 798.917,A -85,B 0,C 180,E1 -10860.113,E2 -10860.113} C_VEL
LIN {X 0,Y 404.683,Z 807.217,A -85,B 0,C 180,E1 -10863.714,E2 -10863.714} C_VEL
LIN {X 0,Y 404.136,Z 815.39,A -85,B 0,C 180,E1 -10867.174,E2 -10867.174} C_VEL
LIN {X 0,Y 403.703,Z 823.856,A -85,B 0,C 180,E1 -10870.685,E2 -10870.685} C_VEL
LIN {X 0,Y 403.532,Z 827.446,A -85,B 0,C 180,E1 -10872.157,E2 -10872.157} C_VEL
LIN {X 0,Y 406.098,Z 845.605,A -85,B 0,C 180,E1 -10873.07,E2 -10873.07} C_VEL
LIN {X 0,Y 407.424,Z 857.484,A -85,B 0,C 180,E1 -10873.766,E2 -10873.766} C_VEL
LIN {X 0,Y 406.67,Z 869.299,A -85,B 0,C 180,E1 -10874.591,E2 -10874.591} C_VEL
LIN {X 0,Y 405.908,Z 880.54,A -85,B 0,C 180,E1 -10875.588,E2 -10875.588} C_VEL
LIN {X 0,Y 405.21,Z 891.049,A -85,B 0,C 180,E1 -10876.744,E2 -10876.744} C_VEL
LIN {X 0,Y 404.583,Z 900.099,A -85,B 0,C 180,E1 -10877.968,E2 -10877.968} C_VEL
LIN {X 0,Y 403.882,Z 909.132,A -85,B 0,C 180,E1 -10879.472,E2 -10879.472} C_VEL
LIN {X 0,Y 403.436,Z 916.431,A -85,B 0,C 180,E1 -10880.98,E2 -10880.98} C_VEL
LIN {X 0,Y 403.182,Z 922.258,A -85,B 0,C 180,E1 -10882.488,E2 -10882.488} C_VEL
LIN {X 0,Y 402.998,Z 926.821,A -85,B 0,C 180,E1 -10883.994,E2 -10883.994} C_VEL
LIN {X 0,Y 403.027,Z 929.22,A -85,B 0,C 180,E1 -10884.998,E2 -10884.998} C_VEL
LIN {X 0,Y 402.894,Z 931.162,A -85,B 0,C 180,E1 -10885.999,E2 -10885.999} C_VEL
LIN {X 0,Y 402.922,Z 932.674,A -85,B 0,C 180,E1 -10887,E2 -10887} C_VEL
LIN {X 0,Y 402.973,Z 933.713,A -85,B 0,C 180,E1 -10888.001,E2 -10888.001} C_VEL
LIN {X 0,Y 402.958,Z 934.337,A -85,B 0,C 180,E1 -10889.001,E2 -10889.001} C_VEL
LIN {X 0,Y 402.979,Z 934.556,A -85,B 0,C 180,E1 -10890,E2 -10890} C_VEL
LIN {X 0,Y 402.958,Z 934.343,A -85,B 0,C 180,E1 -10890.999,E2 -10890.999} C_VEL
LIN {X 0,Y 402.976,Z 933.683,A -85,B 0,C 180,E1 -10891.999,E2 -10891.999} C_VEL
LIN {X 0,Y 402.941,Z 932.614,A -85,B 0,C 180,E1 -10892.999,E2 -10892.999} C_VEL
LIN {X 0,Y 402.911,Z 931.133,A -85,B 0,C 180,E1 -10894.001,E2 -10894.001} C_VEL
LIN {X 0,Y 403.007,Z 928.04,A -85,B 0,C 180,E1 -10895.504,E2 -10895.504} C_VEL
LIN {X 0,Y 403.096,Z 923.87,A -85,B 0,C 180,E1 -10897.01,E2 -10897.01} C_VEL
LIN {X 0,Y 403.414,Z 917.495,A -85,B 0,C 180,E1 -10898.768,E2 -10898.768} C_VEL
LIN {X 0,Y 403.796,Z 910.553,A -85,B 0,C 180,E1 -10900.277,E2 -10900.277} C_VEL
LIN {X 0,Y 404.433,Z 902.029,A -85,B 0,C 180,E1 -10901.782,E2 -10901.782} C_VEL
LIN {X 0,Y 405.067,Z 893.378,A -85,B 0,C 180,E1 -10903.035,E2 -10903.035} C_VEL
LIN {X 0,Y 405.915,Z 882.02,A -85,B 0,C 180,E1 -10904.373,E2 -10904.373} C_VEL
LIN {X 0,Y 406.812,Z 871.201,A -85,B 0,C 180,E1 -10905.404,E2 -10905.404} C_VEL
LIN {X 0,Y 407.665,Z 859.884,A -85,B 0,C 180,E1 -10906.269,E2 -10906.269} C_VEL
LIN {X 0,Y 407.035,Z 850.068,A -85,B 0,C 180,E1 -10906.94,E2 -10906.94} C_VEL
LIN {X 0,Y 405.621,Z 836.075,A -85,B 0,C 180,E1 -10907.724,E2 -10907.724} C_VEL
LIN {X 0,Y 403.52,Z 824.605,A -85,B 0,C 180,E1 -10908.27,E2 -10908.27} C_VEL
LIN {X 0,Y 403.888,Z 815.549,A -85,B 0,C 180,E1 -10911.97,E2 -10911.97} C_VEL
LIN {X 0,Y 404.352,Z 807.699,A -85,B 0,C 180,E1 -10915.336,E2 -10915.336} C_VEL
LIN {X 0,Y 404.844,Z 800.756,A -85,B 0,C 180,E1 -10918.515,E2 -10918.515} C_VEL
LIN {X 0,Y 405.618,Z 793.965,A -85,B 0,C 180,E1 -10921.895,E2 -10921.895} C_VEL
LIN {X 0,Y 406.13,Z 790.424,A -85,B 0,C 180,E1 -10923.835,E2 -10923.835} C_VEL
LIN {X 0,Y 406.411,Z 786.864,A -85,B 0,C 180,E1 -10926.012,E2 -10926.012} C_VEL
LIN {X 0,Y 406.417,Z 784.982,A -85,B 0,C 180,E1 -10927.3,E2 -10927.3} C_VEL
LIN {X 0,Y 406.038,Z 781.882,A -85,B 0,C 180,E1 -10929.824,E2 -10929.824} C_VEL
LIN {X 0,Y 405.62,Z 779.31,A -85,B 0,C 180,E1 -10932.512,E2 -10932.512} C_VEL
LIN {X 0,Y 405.245,Z 777.429,A -85,B 0,C 180,E1 -10935.32,E2 -10935.32} C_VEL
LIN {X 0,Y 405.028,Z 776.154,A -85,B 0,C 180,E1 -10938.747,E2 -10938.747} C_VEL
LIN {X 0,Y 404.919,Z 775.881,A -85,B 0,C 180,E1 -10941.357,E2 -10941.357} C_VEL
LIN {X 0,Y 404.816,Z 776.244,A -85,B 0,C 180,E1 -10944.683,E2 -10944.683} C_VEL
LIN {X 0,Y 404.594,Z 777.06,A -85,B 0,C 180,E1 -10947.418,E2 -10947.418} C_VEL
LIN {X 0,Y 404.239,Z 778.584,A -85,B 0,C 180,E1 -10950.869,E2 -10950.869} C_VEL
LIN {X 0,Y 403.969,Z 780.445,A -85,B 0,C 180,E1 -10954.218,E2 -10954.218} C_VEL
LIN {X 0,Y 403.784,Z 782.544,A -85,B 0,C 180,E1 -10957.485,E2 -10957.485} C_VEL
LIN {X 0,Y 403.605,Z 784.829,A -85,B 0,C 180,E1 -10960.679,E2 -10960.679} C_VEL
LIN {X 0,Y 403.545,Z 785.948,A -85,B 0,C 180,E1 -10961.898,E2 -10961.898} C_VEL
LIN {X 0,Y 407.67,Z 798.961,A -85,B 0,C 180,E1 -10962.728,E2 -10962.728} C_VEL
LIN {X 0,Y 409.139,Z 806.781,A -85,B 0,C 180,E1 -10963.258,E2 -10963.258} C_VEL
LIN {X 0,Y 408.255,Z 819.745,A -85,B 0,C 180,E1 -10964.139,E2 -10964.139} C_VEL
LIN {X 0,Y 407.479,Z 831.161,A -85,B 0,C 180,E1 -10965.142,E2 -10965.142} C_VEL
LIN {X 0,Y 406.501,Z 842.411,A -85,B 0,C 180,E1 -10966.374,E2 -10966.374} C_VEL
LIN {X 0,Y 405.76,Z 850.76,A -85,B 0,C 180,E1 -10967.495,E2 -10967.495} C_VEL
LIN {X 0,Y 405.169,Z 858.479,A -85,B 0,C 180,E1 -10968.746,E2 -10968.746} C_VEL
LIN {X 0,Y 404.491,Z 866.072,A -85,B 0,C 180,E1 -10970.246,E2 -10970.246} C_VEL
LIN {X 0,Y 403.859,Z 873.02,A -85,B 0,C 180,E1 -10971.996,E2 -10971.996} C_VEL
LIN {X 0,Y 403.623,Z 877.143,A -85,B 0,C 180,E1 -10973.32,E2 -10973.32} C_VEL
LIN {X 0,Y 403.222,Z 881.175,A -85,B 0,C 180,E1 -10974.999,E2 -10974.999} C_VEL
LIN {X 0,Y 403.259,Z 882.961,A -85,B 0,C 180,E1 -10976.002,E2 -10976.002} C_VEL
LIN {X 0,Y 403.124,Z 884.289,A -85,B 0,C 180,E1 -10977.001,E2 -10977.001} C_VEL
LIN {X 0,Y 403.062,Z 885.208,A -85,B 0,C 180,E1 -10978.001,E2 -10978.001} C_VEL
LIN {X 0,Y 403.016,Z 885.735,A -85,B 0,C 180,E1 -10979,E2 -10979} C_VEL
LIN {X 0,Y 402.979,Z 885.85,A -85,B 0,C 180,E1 -10979.999,E2 -10979.999} C_VEL
LIN {X 0,Y 402.988,Z 885.529,A -85,B 0,C 180,E1 -10980.998,E2 -10980.998} C_VEL
LIN {X 0,Y 403.034,Z 884.815,A -85,B 0,C 180,E1 -10981.998,E2 -10981.998} C_VEL
LIN {X 0,Y 403.096,Z 883.704,A -85,B 0,C 180,E1 -10982.997,E2 -10982.997} C_VEL
LIN {X 0,Y 403.124,Z 882.151,A -85,B 0,C 180,E1 -10983.998,E2 -10983.998} C_VEL
LIN {X 0,Y 403.247,Z 879.004,A -85,B 0,C 180,E1 -10985.5,E2 -10985.5} C_VEL
LIN {X 0,Y 403.451,Z 874.78,A -85,B 0,C 180,E1 -10987.003,E2 -10987.003} C_VEL
LIN {X 0,Y 403.876,Z 868.331,A -85,B 0,C 180,E1 -10988.757,E2 -10988.757} C_VEL
LIN {X 0,Y 404.372,Z 861.325,A -85,B 0,C 180,E1 -10990.261,E2 -10990.261} C_VEL
LIN {X 0,Y 404.992,Z 852.565,A -85,B 0,C 180,E1 -10991.764,E2 -10991.764} C_VEL
LIN {X 0,Y 405.721,Z 843.623,A -85,B 0,C 180,E1 -10993.013,E2 -10993.013} C_VEL
LIN {X 0,Y 406.415,Z 833.594,A -85,B 0,C 180,E1 -10994.166,E2 -10994.166} C_VEL
LIN {X 0,Y 407.04,Z 823.21,A -85,B 0,C 180,E1 -10995.137,E2 -10995.137} C_VEL
LIN {X 0,Y 407.745,Z 811.494,A -85,B 0,C 180,E1 -10996.007,E2 -10996.007} C_VEL
LIN {X 0,Y 408.009,Z 804.253,A -85,B 0,C 180,E1 -10996.452,E2 -10996.452} C_VEL
LIN {X 0,Y 405.448,Z 792.109,A -85,B 0,C 180,E1 -10997.15,E2 -10997.15} C_VEL
LIN {X 0,Y 403.092,Z 782.04,A -85,B 0,C 180,E1 -10997.619,E2 -10997.619} C_VEL
LIN {X 0,Y 403.099,Z 779.217,A -85,B 0,C 180,E1 -11000.406,E2 -11000.406} C_VEL
LIN {X 0,Y 403.178,Z 776.009,A -85,B 0,C 180,E1 -11003.635,E2 -11003.635} C_VEL
LIN {X 0,Y 403.32,Z 772.792,A -85,B 0,C 180,E1 -11006.939,E2 -11006.939} C_VEL
LIN {X 0,Y 403.294,Z 771.707,A -85,B 0,C 180,E1 -11008.066,E2 -11008.066} C_VEL
LIN {X 0,Y 403.425,Z 771.234,A -85,B 0,C 180,E1 -11009.42,E2 -11009.42} C_VEL
LIN {X 0,Y 403.82,Z 771.186,A -85,B 0,C 180,E1 -11012.649,E2 -11012.649} C_VEL
LIN {X 0,Y 404.048,Z 771.154,A -85,B 0,C 180,E1 -11015.163,E2 -11015.163} C_VEL
LIN {X 0,Y 404.148,Z 771.143,A -85,B 0,C 180,E1 -11018.506,E2 -11018.506} C_VEL
LIN {X 0,Y 404.118,Z 771.145,A -85,B 0,C 180,E1 -11021.599,E2 -11021.599} C_VEL
LIN {X 0,Y 404.14,Z 771.143,A -85,B 0,C 180,E1 -11024.521,E2 -11024.521} C_VEL
LIN {X 0,Y 404.131,Z 771.145,A -85,B 0,C 180,E1 -11027.295,E2 -11027.295} C_VEL
LIN {X 0,Y 404.163,Z 771.139,A -85,B 0,C 180,E1 -11029.954,E2 -11029.954} C_VEL
LIN {X 0,Y 404.129,Z 771.147,A -85,B 0,C 180,E1 -11033.124,E2 -11033.124} C_VEL
LIN {X 0,Y 404.137,Z 771.142,A -85,B 0,C 180,E1 -11036.187,E2 -11036.187} C_VEL
LIN {X 0,Y 404.136,Z 771.143,A -85,B 0,C 180,E1 -11039.714,E2 -11039.714} C_VEL
LIN {X 0,Y 404.127,Z 771.145,A -85,B 0,C 180,E1 -11043.118,E2 -11043.118} C_VEL
LIN {X 0,Y 404.151,Z 771.139,A -85,B 0,C 180,E1 -11046.424,E2 -11046.424} C_VEL
LIN {X 0,Y 404.182,Z 771.138,A -85,B 0,C 180,E1 -11049.874,E2 -11049.874} C_VEL
LIN {X 0,Y 404.207,Z 771.133,A -85,B 0,C 180,E1 -11052.993,E2 -11052.993} C_VEL
LIN {X 0,Y 404.274,Z 771.124,A -85,B 0,C 180,E1 -11056.939,E2 -11056.939} C_VEL
LIN {X 0,Y 404.244,Z 771.131,A -85,B 0,C 180,E1 -11059.988,E2 -11059.988} C_VEL
LIN {X 0,Y 404.33,Z 771.116,A -85,B 0,C 180,E1 -11063.011,E2 -11063.011} C_VEL
LIN {X 0,Y 404.246,Z 771.127,A -85,B 0,C 180,E1 -11065.013,E2 -11065.013} C_VEL
LIN {X 0,Y 404.46,Z 771.107,A -85,B 0,C 180,E1 -11068.008,E2 -11068.008} C_VEL
LIN {X 0,Y 404.336,Z 771.115,A -85,B 0,C 180,E1 -11070.996,E2 -11070.996} C_VEL
LIN {X 0,Y 404.347,Z 771.113,A -85,B 0,C 180,E1 -11072.989,E2 -11072.989} C_VEL
LIN {X 0,Y 404.355,Z 771.118,A -85,B 0,C 180,E1 -11075.986,E2 -11075.986} C_VEL
LIN {X 0,Y 404.244,Z 771.127,A -85,B 0,C 180,E1 -11079.002,E2 -11079.002} C_VEL
LIN {X 0,Y 404.238,Z 771.131,A -85,B 0,C 180,E1 -11082.042,E2 -11082.042} C_VEL
LIN {X 0,Y 404.195,Z 771.133,A -85,B 0,C 180,E1 -11085.118,E2 -11085.118} C_VEL
LIN {X 0,Y 404.179,Z 771.136,A -85,B 0,C 180,E1 -11087.917,E2 -11087.917} C_VEL
LIN {X 0,Y 403.526,Z 771.223,A -85,B 0,C 180,E1 -11088.749,E2 -11088.749} C_VEL
LIN {X 0,Y 400.647,Z 771.579,A -85,B 0,C 180,E1 -11090.101,E2 -11090.101} C_VEL
LIN {X 0,Y 398.201,Z 771.881,A -85,B 0,C 180,E1 -11091.193,E2 -11091.193} C_VEL
LIN {X 0,Y 397.154,Z 772.012,A -85,B 0,C 180,E1 -11092.037,E2 -11092.037} C_VEL
LIN {X 0,Y 397.072,Z 772.02,A -85,B 0,C 180,E1 -11092.323,E2 -11092.323} C_VEL
LIN {X 0,Y 397.087,Z 772.019,A -85,B 0,C 180,E1 -11095.496,E2 -11095.496} C_VEL
LIN {X 0,Y 397.07,Z 772.026,A -85,B 0,C 180,E1 -11098.548,E2 -11098.548} C_VEL
LIN {X 0,Y 397.073,Z 772.021,A -85,B 0,C 180,E1 -11101.837,E2 -11101.837} C_VEL
LIN {X 0,Y 397.117,Z 772.018,A -85,B 0,C 180,E1 -11104.494,E2 -11104.494} C_VEL
LIN {X 0,Y 397.094,Z 772.019,A -85,B 0,C 180,E1 -11108.276,E2 -11108.276} C_VEL
LIN {X 0,Y 397.082,Z 772.025,A -85,B 0,C 180,E1 -11110.91,E2 -11110.91} C_VEL
LIN {X 0,Y 397.095,Z 772.02,A -85,B 0,C 180,E1 -11113.65,E2 -11113.65} C_VEL
LIN {X 0,Y 397.097,Z 772.019,A -85,B 0,C 180,E1 -11116.522,E2 -11116.522} C_VEL
LIN {X 0,Y 397.109,Z 772.017,A -85,B 0,C 180,E1 -11120.424,E2 -11120.424} C_VEL
LIN {X 0,Y 397.084,Z 772.023,A -85,B 0,C 180,E1 -11123.005,E2 -11123.005} C_VEL
LIN {X 0,Y 396.905,Z 772.044,A -85,B 0,C 180,E1 -11126.329,E2 -11126.329} C_VEL
LIN {X 0,Y 396.563,Z 772.088,A -85,B 0,C 180,E1 -11129.074,E2 -11129.074} C_VEL
LIN {X 0,Y 396.182,Z 772.137,A -85,B 0,C 180,E1 -11132.535,E2 -11132.535} C_VEL
LIN {X 0,Y 396.125,Z 772.914,A -85,B 0,C 180,E1 -11133.671,E2 -11133.671} C_VEL
LIN {X 0,Y 396.046,Z 776.815,A -85,B 0,C 180,E1 -11137.334,E2 -11137.334} C_VEL
LIN {X 0,Y 396.049,Z 779.978,A -85,B 0,C 180,E1 -11140.297,E2 -11140.297} C_VEL
LIN {X 0,Y 395.992,Z 782.07,A -85,B 0,C 180,E1 -11142.241,E2 -11142.241} C_VEL
LIN {X 0,Y 399.014,Z 795.279,A -85,B 0,C 180,E1 -11142.874,E2 -11142.874} C_VEL
LIN {X 0,Y 401.054,Z 805.604,A -85,B 0,C 180,E1 -11143.501,E2 -11143.501} C_VEL
LIN {X 0,Y 400.374,Z 818.091,A -85,B 0,C 180,E1 -11144.344,E2 -11144.344} C_VEL
LIN {X 0,Y 399.626,Z 830.384,A -85,B 0,C 180,E1 -11145.411,E2 -11145.411} C_VEL
LIN {X 0,Y 398.889,Z 841.427,A -85,B 0,C 180,E1 -11146.631,E2 -11146.631} C_VEL
LIN {X 0,Y 398.047,Z 851.684,A -85,B 0,C 180,E1 -11148.028,E2 -11148.028} C_VEL
LIN {X 0,Y 397.393,Z 860.633,A -85,B 0,C 180,E1 -11149.557,E2 -11149.557} C_VEL
LIN {X 0,Y 396.82,Z 867.876,A -85,B 0,C 180,E1 -11151.086,E2 -11151.086} C_VEL
LIN {X 0,Y 396.503,Z 872.768,A -85,B 0,C 180,E1 -11152.362,E2 -11152.362} C_VEL
LIN {X 0,Y 396.301,Z 877.519,A -85,B 0,C 180,E1 -11153.893,E2 -11153.893} C_VEL
LIN {X 0,Y 396.016,Z 881.145,A -85,B 0,C 180,E1 -11155.421,E2 -11155.421} C_VEL
LIN {X 0,Y 396.009,Z 883.733,A -85,B 0,C 180,E1 -11156.949,E2 -11156.949} C_VEL
LIN {X 0,Y 395.954,Z 884.924,A -85,B 0,C 180,E1 -11157.967,E2 -11157.967} C_VEL
LIN {X 0,Y 395.875,Z 886.058,A -85,B 0,C 180,E1 -11160.001,E2 -11160.001} C_VEL
LIN {X 0,Y 395.924,Z 886.024,A -85,B 0,C 180,E1 -11161.018,E2 -11161.018} C_VEL
LIN {X 0,Y 395.968,Z 885.541,A -85,B 0,C 180,E1 -11162.035,E2 -11162.035} C_VEL
LIN {X 0,Y 396.192,Z 883.389,A -85,B 0,C 180,E1 -11164.07,E2 -11164.07} C_VEL
LIN {X 0,Y 396.227,Z 880.658,A -85,B 0,C 180,E1 -11165.599,E2 -11165.599} C_VEL
LIN {X 0,Y 396.633,Z 876.872,A -85,B 0,C 180,E1 -11167.126,E2 -11167.126} C_VEL
LIN {X 0,Y 396.984,Z 871.951,A -85,B 0,C 180,E1 -11168.656,E2 -11168.656} C_VEL
LIN {X 0,Y 397.556,Z 865.706,A -85,B 0,C 180,E1 -11170.183,E2 -11170.183} C_VEL
LIN {X 0,Y 398.329,Z 857.941,A -85,B 0,C 180,E1 -11171.708,E2 -11171.708} C_VEL
LIN {X 0,Y 398.964,Z 850.088,A -85,B 0,C 180,E1 -11172.98,E2 -11172.98} C_VEL
LIN {X 0,Y 399.888,Z 840.546,A -85,B 0,C 180,E1 -11174.245,E2 -11174.245} C_VEL
LIN {X 0,Y 400.708,Z 830.008,A -85,B 0,C 180,E1 -11175.384,E2 -11175.384} C_VEL
LIN {X 0,Y 401.688,Z 818.403,A -85,B 0,C 180,E1 -11176.385,E2 -11176.385} C_VEL
LIN {X 0,Y 402.419,Z 807.402,A -85,B 0,C 180,E1 -11177.131,E2 -11177.131} C_VEL
LIN {X 0,Y 399.955,Z 796.351,A -85,B 0,C 180,E1 -11177.916,E2 -11177.916} C_VEL
LIN {X 0,Y 396.382,Z 785.278,A -85,B 0,C 180,E1 -11178.646,E2 -11178.646} C_VEL
LIN {X 0,Y 396.402,Z 783.087,A -85,B 0,C 180,E1 -11180.769,E2 -11180.769} C_VEL
LIN {X 0,Y 396.504,Z 779.648,A -85,B 0,C 180,E1 -11184.06,E2 -11184.06} C_VEL
LIN {X 0,Y 396.588,Z 775.852,A -85,B 0,C 180,E1 -11187.618,E2 -11187.618} C_VEL
LIN {X 0,Y 396.571,Z 772.27,A -85,B 0,C 180,E1 -11190.927,E2 -11190.927} C_VEL
LIN {X 0,Y 396.897,Z 772.049,A -85,B 0,C 180,E1 -11193.669,E2 -11193.669} C_VEL
LIN {X 0,Y 397.09,Z 772.024,A -85,B 0,C 180,E1 -11196.997,E2 -11196.997} C_VEL
LIN {X 0,Y 397.107,Z 772.02,A -85,B 0,C 180,E1 -11199.579,E2 -11199.579} C_VEL
LIN {X 0,Y 397.105,Z 772.02,A -85,B 0,C 180,E1 -11203.479,E2 -11203.479} C_VEL
LIN {X 0,Y 397.124,Z 772.123,A -85,B 0,C 180,E1 -11206.424,E2 -11206.424} C_VEL
LIN {X 0,Y 398.107,Z 777.569,A -85,B 0,C 180,E1 -11209.386,E2 -11209.386} C_VEL
LIN {X 0,Y 399.132,Z 783.395,A -85,B 0,C 180,E1 -11212.409,E2 -11212.409} C_VEL
LIN {X 0,Y 399.342,Z 787.635,A -85,B 0,C 180,E1 -11214.495,E2 -11214.495} C_VEL
LIN {X 0,Y 398.73,Z 794.698,A -85,B 0,C 180,E1 -11217.785,E2 -11217.785} C_VEL
LIN {X 0,Y 398.068,Z 801.715,A -85,B 0,C 180,E1 -11220.953,E2 -11220.953} C_VEL
LIN {X 0,Y 397.493,Z 809.507,A -85,B 0,C 180,E1 -11224.387,E2 -11224.387} C_VEL
LIN {X 0,Y 396.996,Z 817.04,A -85,B 0,C 180,E1 -11227.628,E2 -11227.628} C_VEL
LIN {X 0,Y 396.588,Z 824.687,A -85,B 0,C 180,E1 -11230.862,E2 -11230.862} C_VEL
LIN {X 0,Y 396.488,Z 826.885,A -85,B 0,C 180,E1 -11231.729,E2 -11231.729} C_VEL
LIN {X 0,Y 398.164,Z 837.193,A -85,B 0,C 180,E1 -11232.249,E2 -11232.249} C_VEL
LIN {X 0,Y 399.682,Z 850.706,A -85,B 0,C 180,E1 -11233.068,E2 -11233.068} C_VEL
LIN {X 0,Y 400.418,Z 859.59,A -85,B 0,C 180,E1 -11233.69,E2 -11233.69} C_VEL
LIN {X 0,Y 399.557,Z 871.338,A -85,B 0,C 180,E1 -11234.571,E2 -11234.571} C_VEL
LIN {X 0,Y 398.787,Z 882.108,A -85,B 0,C 180,E1 -11235.586,E2 -11235.586} C_VEL
LIN {X 0,Y 398.119,Z 891.964,A -85,B 0,C 180,E1 -11236.733,E2 -11236.733} C_VEL
LIN {X 0,Y 397.443,Z 900.963,A -85,B 0,C 180,E1 -11238.008,E2 -11238.008} C_VEL
LIN {X 0,Y 396.779,Z 909.789,A -85,B 0,C 180,E1 -11239.54,E2 -11239.54} C_VEL
LIN {X 0,Y 396.349,Z 916.849,A -85,B 0,C 180,E1 -11241.074,E2 -11241.074} C_VEL
LIN {X 0,Y 396.028,Z 923.304,A -85,B 0,C 180,E1 -11242.864,E2 -11242.864} C_VEL
LIN {X 0,Y 395.916,Z 927.527,A -85,B 0,C 180,E1 -11244.397,E2 -11244.397} C_VEL
LIN {X 0,Y 395.819,Z 930.643,A -85,B 0,C 180,E1 -11245.927,E2 -11245.927} C_VEL
LIN {X 0,Y 395.829,Z 932.176,A -85,B 0,C 180,E1 -11246.947,E2 -11246.947} C_VEL
LIN {X 0,Y 395.902,Z 933.238,A -85,B 0,C 180,E1 -11247.965,E2 -11247.965} C_VEL
LIN {X 0,Y 395.882,Z 933.872,A -85,B 0,C 180,E1 -11248.983,E2 -11248.983} C_VEL
LIN {X 0,Y 395.9,Z 934.104,A -85,B 0,C 180,E1 -11250,E2 -11250} C_VEL
LIN {X 0,Y 395.883,Z 933.915,A -85,B 0,C 180,E1 -11251.017,E2 -11251.017} C_VEL
LIN {X 0,Y 395.906,Z 933.268,A -85,B 0,C 180,E1 -11252.035,E2 -11252.035} C_VEL
LIN {X 0,Y 395.844,Z 932.202,A -85,B 0,C 180,E1 -11253.053,E2 -11253.053} C_VEL
LIN {X 0,Y 395.833,Z 930.73,A -85,B 0,C 180,E1 -11254.073,E2 -11254.073} C_VEL
LIN {X 0,Y 395.906,Z 927.648,A -85,B 0,C 180,E1 -11255.603,E2 -11255.603} C_VEL
LIN {X 0,Y 396.024,Z 923.491,A -85,B 0,C 180,E1 -11257.136,E2 -11257.136} C_VEL
LIN {X 0,Y 396.368,Z 917.166,A -85,B 0,C 180,E1 -11258.925,E2 -11258.925} C_VEL
LIN {X 0,Y 396.768,Z 910.284,A -85,B 0,C 180,E1 -11260.461,E2 -11260.461} C_VEL
LIN {X 0,Y 397.448,Z 901.809,A -85,B 0,C 180,E1 -11261.992,E2 -11261.992} C_VEL
LIN {X 0,Y 398.13,Z 893.219,A -85,B 0,C 180,E1 -11263.267,E2 -11263.267} C_VEL
LIN {X 0,Y 398.953,Z 882.754,A -85,B 0,C 180,E1 -11264.538,E2 -11264.538} C_VEL
LIN {X 0,Y 399.968,Z 871.297,A -85,B 0,C 180,E1 -11265.674,E2 -11265.674} C_VEL
LIN {X 0,Y 400.874,Z 860.317,A -85,B 0,C 180,E1 -11266.552,E2 -11266.552} C_VEL
LIN {X 0,Y 400.001,Z 847.393,A -85,B 0,C 180,E1 -11267.451,E2 -11267.451} C_VEL
LIN {X 0,Y 398.522,Z 834.392,A -85,B 0,C 180,E1 -11268.193,E2 -11268.193} C_VEL
LIN {X 0,Y 396.462,Z 823.965,A -85,B 0,C 180,E1 -11268.742,E2 -11268.742} C_VEL
LIN {X 0,Y 396.864,Z 815.3,A -85,B 0,C 180,E1 -11272.38,E2 -11272.38} C_VEL
LIN {X 0,Y 397.335,Z 808.094,A -85,B 0,C 180,E1 -11275.566,E2 -11275.566} C_VEL
LIN {X 0,Y 397.935,Z 800.716,A -85,B 0,C 180,E1 -11279.057,E2 -11279.057} C_VEL
LIN {X 0,Y 398.695,Z 794.638,A -85,B 0,C 180,E1 -11282.207,E2 -11282.207} C_VEL
LIN {X 0,Y 399.216,Z 790.992,A -85,B 0,C 180,E1 -11284.288,E2 -11284.288} C_VEL
LIN {X 0,Y 399.445,Z 787.22,A -85,B 0,C 180,E1 -11286.742,E2 -11286.742} C_VEL
LIN {X 0,Y 399.183,Z 783.933,A -85,B 0,C 180,E1 -11289.332,E2 -11289.332} C_VEL
LIN {X 0,Y 398.741,Z 781.07,A -85,B 0,C 180,E1 -11292.245,E2 -11292.245} C_VEL
LIN {X 0,Y 398.361,Z 779.084,A -85,B 0,C 180,E1 -11295.114,E2 -11295.114} C_VEL
LIN {X 0,Y 398.13,Z 777.913,A -85,B 0,C 180,E1 -11297.871,E2 -11297.871} C_VEL
LIN {X 0,Y 397.992,Z 777.364,A -85,B 0,C 180,E1 -11300.985,E2 -11300.985} C_VEL
LIN {X 0,Y 397.905,Z 777.407,A -85,B 0,C 180,E1 -11303.091,E2 -11303.091} C_VEL
LIN {X 0,Y 397.745,Z 777.978,A -85,B 0,C 180,E1 -11306.148,E2 -11306.148} C_VEL
LIN {X 0,Y 397.4,Z 779.036,A -85,B 0,C 180,E1 -11309.144,E2 -11309.144} C_VEL
LIN {X 0,Y 397.097,Z 780.684,A -85,B 0,C 180,E1 -11312.602,E2 -11312.602} C_VEL
LIN {X 0,Y 396.817,Z 782.648,A -85,B 0,C 180,E1 -11315.96,E2 -11315.96} C_VEL
LIN {X 0,Y 396.651,Z 784.82,A -85,B 0,C 180,E1 -11319.244,E2 -11319.244} C_VEL
LIN {X 0,Y 396.504,Z 786.401,A -85,B 0,C 180,E1 -11321.423,E2 -11321.423} C_VEL
LIN {X 0,Y 400.637,Z 799.103,A -85,B 0,C 180,E1 -11322.3,E2 -11322.3} C_VEL
LIN {X 0,Y 402.465,Z 807.182,A -85,B 0,C 180,E1 -11322.885,E2 -11322.885} C_VEL
LIN {X 0,Y 401.66,Z 819.569,A -85,B 0,C 180,E1 -11323.741,E2 -11323.741} C_VEL
LIN {X 0,Y 400.832,Z 831.024,A -85,B 0,C 180,E1 -11324.751,E2 -11324.751} C_VEL
LIN {X 0,Y 399.823,Z 842.384,A -85,B 0,C 180,E1 -11326.012,E2 -11326.012} C_VEL
LIN {X 0,Y 398.891,Z 851.621,A -85,B 0,C 180,E1 -11327.276,E2 -11327.276} C_VEL
LIN {X 0,Y 398.116,Z 860.625,A -85,B 0,C 180,E1 -11328.802,E2 -11328.802} C_VEL
LIN {X 0,Y 397.443,Z 867.877,A -85,B 0,C 180,E1 -11330.328,E2 -11330.328} C_VEL
LIN {X 0,Y 396.875,Z 873.697,A -85,B 0,C 180,E1 -11331.855,E2 -11331.855} C_VEL
LIN {X 0,Y 396.589,Z 877.95,A -85,B 0,C 180,E1 -11333.268,E2 -11333.268} C_VEL
LIN {X 0,Y 396.165,Z 881.748,A -85,B 0,C 180,E1 -11334.91,E2 -11334.91} C_VEL
LIN {X 0,Y 396.208,Z 883.496,A -85,B 0,C 180,E1 -11335.93,E2 -11335.93} C_VEL
LIN {X 0,Y 395.991,Z 885.697,A -85,B 0,C 180,E1 -11337.965,E2 -11337.965} C_VEL
LIN {X 0,Y 395.938,Z 886.208,A -85,B 0,C 180,E1 -11338.982,E2 -11338.982} C_VEL
LIN {X 0,Y 395.9,Z 886.29,A -85,B 0,C 180,E1 -11339.999,E2 -11339.999} C_VEL
LIN {X 0,Y 395.911,Z 885.947,A -85,B 0,C 180,E1 -11341.016,E2 -11341.016} C_VEL
LIN {X 0,Y 395.965,Z 885.208,A -85,B 0,C 180,E1 -11342.033,E2 -11342.033} C_VEL
LIN {X 0,Y 396.037,Z 884.072,A -85,B 0,C 180,E1 -11343.051,E2 -11343.051} C_VEL
LIN {X 0,Y 396.036,Z 881.542,A -85,B 0,C 180,E1 -11344.579,E2 -11344.579} C_VEL
LIN {X 0,Y 396.369,Z 876.926,A -85,B 0,C 180,E1 -11346.486,E2 -11346.486} C_VEL
LIN {X 0,Y 396.62,Z 871.491,A -85,B 0,C 180,E1 -11348.148,E2 -11348.148} C_VEL
LIN {X 0,Y 397.109,Z 865.137,A -85,B 0,C 180,E1 -11349.678,E2 -11349.678} C_VEL
LIN {X 0,Y 397.712,Z 857.212,A -85,B 0,C 180,E1 -11351.207,E2 -11351.207} C_VEL
LIN {X 0,Y 398.301,Z 849.143,A -85,B 0,C 180,E1 -11352.482,E2 -11352.482} C_VEL
LIN {X 0,Y 399.135,Z 839.358,A -85,B 0,C 180,E1 -11353.75,E2 -11353.75} C_VEL
LIN {X 0,Y 399.783,Z 828.629,A -85,B 0,C 180,E1 -11354.888,E2 -11354.888} C_VEL
LIN {X 0,Y 400.553,Z 816.385,A -85,B 0,C 180,E1 -11355.91,E2 -11355.91} C_VEL
LIN {X 0,Y 401.121,Z 805.784,A -85,B 0,C 180,E1 -11356.61,E2 -11356.61} C_VEL
LIN {X 0,Y 398.826,Z 794.398,A -85,B 0,C 180,E1 -11357.299,E2 -11357.299} C_VEL
LIN {X 0,Y 395.988,Z 782.411,A -85,B 0,C 180,E1 -11357.873,E2 -11357.873} C_VEL
LIN {X 0,Y 396.027,Z 779.48,A -85,B 0,C 180,E1 -11360.788,E2 -11360.788} C_VEL
LIN {X 0,Y 396.119,Z 777.309,A -85,B 0,C 180,E1 -11362.974,E2 -11362.974} C_VEL
LIN {X 0,Y 396.209,Z 774.07,A -85,B 0,C 180,E1 -11366.323,E2 -11366.323} C_VEL
LIN {X 0,Y 396.272,Z 772.126,A -85,B 0,C 180,E1 -11368.609,E2 -11368.609} C_VEL
LIN {X 0,Y 396.701,Z 772.073,A -85,B 0,C 180,E1 -11372.104,E2 -11372.104} C_VEL
LIN {X 0,Y 396.941,Z 772.044,A -85,B 0,C 180,E1 -11374.51,E2 -11374.51} C_VEL
LIN {X 0,Y 397.079,Z 772.022,A -85,B 0,C 180,E1 -11377.206,E2 -11377.206} C_VEL
LIN {X 0,Y 397.097,Z 772.021,A -85,B 0,C 180,E1 -11380.444,E2 -11380.444} C_VEL
LIN {X 0,Y 397.096,Z 772.019,A -85,B 0,C 180,E1 -11383.647,E2 -11383.647} C_VEL
LIN {X 0,Y 397.096,Z 772.021,A -85,B 0,C 180,E1 -11386.52,E2 -11386.52} C_VEL
LIN {X 0,Y 397.107,Z 772.019,A -85,B 0,C 180,E1 -11390.422,E2 -11390.422} C_VEL
LIN {X 0,Y 397.1,Z 772.019,A -85,B 0,C 180,E1 -11394.264,E2 -11394.264} C_VEL
LIN {X 0,Y 397.107,Z 772.019,A -85,B 0,C 180,E1 -11396.726,E2 -11396.726} C_VEL
LIN {X 0,Y 397.11,Z 772.017,A -85,B 0,C 180,E1 -11400.295,E2 -11400.295} C_VEL
LIN {X 0,Y 397.087,Z 772.022,A -85,B 0,C 180,E1 -11403.738,E2 -11403.738} C_VEL
LIN {X 0,Y 397.095,Z 772.02,A -85,B 0,C 180,E1 -11407.085,E2 -11407.085} C_VEL
LIN {X 0,Y 397.137,Z 772.013,A -85,B 0,C 180,E1 -11410.352,E2 -11410.352} C_VEL
LIN {X 0,Y 397.157,Z 772.016,A -85,B 0,C 180,E1 -11413.553,E2 -11413.553} C_VEL
LIN {X 0,Y 397.22,Z 772.002,A -85,B 0,C 180,E1 -11416.702,E2 -11416.702} C_VEL
LIN {X 0,Y 397.204,Z 772.01,A -85,B 0,C 180,E1 -11419.809,E2 -11419.809} C_VEL
LIN {X 0,Y 397.283,Z 771.994,A -85,B 0,C 180,E1 -11422.887,E2 -11422.887} C_VEL
LIN {X 0,Y 397.217,Z 772.002,A -85,B 0,C 180,E1 -11424.925,E2 -11424.925} C_VEL
LIN {X 0,Y 397.428,Z 771.983,A -85,B 0,C 180,E1 -11427.973,E2 -11427.973} C_VEL
LIN {X 0,Y 397.426,Z 771.983,A -85,B 0,C 180,E1 -11432.027,E2 -11432.027} C_VEL
LIN {X 0,Y 397.309,Z 771.997,A -85,B 0,C 180,E1 -11436.093,E2 -11436.093} C_VEL
LIN {X 0,Y 397.216,Z 772.002,A -85,B 0,C 180,E1 -11439.163,E2 -11439.163} C_VEL
LIN {X 0,Y 397.203,Z 772.01,A -85,B 0,C 180,E1 -11442.259,E2 -11442.259} C_VEL
LIN {X 0,Y 397.169,Z 772.008,A -85,B 0,C 180,E1 -11445.393,E2 -11445.393} C_VEL
LIN {X 0,Y 397.148,Z 772.016,A -85,B 0,C 180,E1 -11448.574,E2 -11448.574} C_VEL
LIN {X 0,Y 397.087,Z 772.019,A -85,B 0,C 180,E1 -11451.819,E2 -11451.819} C_VEL
LIN {X 0,Y 397.072,Z 772.02,A -85,B 0,C 180,E1 -11452.323,E2 -11452.323} C_VEL
LIN {X 0,Y 396.424,Z 772.105,A -85,B 0,C 180,E1 -11453.169,E2 -11453.169} C_VEL
LIN {X 0,Y 393.61,Z 772.462,A -85,B 0,C 180,E1 -11454.545,E2 -11454.545} C_VEL
LIN {X 0,Y 391.202,Z 772.764,A -85,B 0,C 180,E1 -11455.657,E2 -11455.657} C_VEL
LIN {X 0,Y 390.141,Z 772.892,A -85,B 0,C 180,E1 -11456.516,E2 -11456.516} C_VEL
LIN {X 0,Y 390.04,Z 772.901,A -85,B 0,C 180,E1 -11456.807,E2 -11456.807} C_VEL
LIN {X 0,Y 390.029,Z 772.9,A -85,B 0,C 180,E1 -11460.301,E2 -11460.301} C_VEL
LIN {X 0,Y 390.061,Z 772.895,A -85,B 0,C 180,E1 -11464.025,E2 -11464.025} C_VEL
LIN {X 0,Y 390.036,Z 772.899,A -85,B 0,C 180,E1 -11467.552,E2 -11467.552} C_VEL
LIN {X 0,Y 390.05,Z 772.9,A -85,B 0,C 180,E1 -11470.822,E2 -11470.822} C_VEL
LIN {X 0,Y 390.049,Z 772.897,A -85,B 0,C 180,E1 -11473.887,E2 -11473.887} C_VEL
LIN {X 0,Y 390.052,Z 772.898,A -85,B 0,C 180,E1 -11476.791,E2 -11476.791} C_VEL
LIN {X 0,Y 390.052,Z 772.898,A -85,B 0,C 180,E1 -11479.562,E2 -11479.562} C_VEL
LIN {X 0,Y 390.034,Z 772.899,A -85,B 0,C 180,E1 -11482.451,E2 -11482.451} C_VEL
LIN {X 0,Y 389.894,Z 772.919,A -85,B 0,C 180,E1 -11486.014,E2 -11486.014} C_VEL
LIN {X 0,Y 389.605,Z 772.953,A -85,B 0,C 180,E1 -11488.459,E2 -11488.459} C_VEL
LIN {X 0,Y 389.175,Z 773.01,A -85,B 0,C 180,E1 -11491.998,E2 -11491.998} C_VEL
LIN {X 0,Y 389.048,Z 773.027,A -85,B 0,C 180,E1 -11493.154,E2 -11493.154} C_VEL
LIN {X 0,Y 388.951,Z 776.633,A -85,B 0,C 180,E1 -11496.578,E2 -11496.578} C_VEL
LIN {X 0,Y 388.982,Z 780.265,A -85,B 0,C 180,E1 -11499.972,E2 -11499.972} C_VEL
LIN {X 0,Y 388.91,Z 782.413,A -85,B 0,C 180,E1 -11501.974,E2 -11501.974} C_VEL
LIN {X 0,Y 391.766,Z 794.988,A -85,B 0,C 180,E1 -11502.583,E2 -11502.583} C_VEL
LIN {X 0,Y 394.132,Z 806.515,A -85,B 0,C 180,E1 -11503.301,E2 -11503.301} C_VEL
LIN {X 0,Y 393.398,Z 819.288,A -85,B 0,C 180,E1 -11504.192,E2 -11504.192} C_VEL
LIN {X 0,Y 392.668,Z 830.89,A -85,B 0,C 180,E1 -11505.227,E2 -11505.227} C_VEL
LIN {X 0,Y 391.868,Z 842.318,A -85,B 0,C 180,E1 -11506.519,E2 -11506.519} C_VEL
LIN {X 0,Y 391.08,Z 851.647,A -85,B 0,C 180,E1 -11507.811,E2 -11507.811} C_VEL
LIN {X 0,Y 390.385,Z 860.688,A -85,B 0,C 180,E1 -11509.368,E2 -11509.368} C_VEL
LIN {X 0,Y 389.803,Z 867.999,A -85,B 0,C 180,E1 -11510.924,E2 -11510.924} C_VEL
LIN {X 0,Y 389.458,Z 872.953,A -85,B 0,C 180,E1 -11512.223,E2 -11512.223} C_VEL
LIN {X 0,Y 389.246,Z 877.76,A -85,B 0,C 180,E1 -11513.782,E2 -11513.782} C_VEL
LIN {X 0,Y 388.947,Z 881.44,A -85,B 0,C 180,E1 -11515.337,E2 -11515.337} C_VEL
LIN {X 0,Y 388.934,Z 884.072,A -85,B 0,C 180,E1 -11516.894,E2 -11516.894} C_VEL
LIN {X 0,Y 388.887,Z 885.303,A -85,B 0,C 180,E1 -11517.93,E2 -11517.93} C_VEL
LIN {X 0,Y 388.826,Z 886.089,A -85,B 0,C 180,E1 -11518.965,E2 -11518.965} C_VEL
LIN {X 0,Y 388.849,Z 886.482,A -85,B 0,C 180,E1 -11521.037,E2 -11521.037} C_VEL
LIN {X 0,Y 388.901,Z 886.033,A -85,B 0,C 180,E1 -11522.072,E2 -11522.072} C_VEL
LIN {X 0,Y 389.003,Z 885.178,A -85,B 0,C 180,E1 -11523.108,E2 -11523.108} C_VEL
LIN {X 0,Y 389.141,Z 883.928,A -85,B 0,C 180,E1 -11524.144,E2 -11524.144} C_VEL
LIN {X 0,Y 389.191,Z 881.236,A -85,B 0,C 180,E1 -11525.701,E2 -11525.701} C_VEL
LIN {X 0,Y 389.619,Z 877.488,A -85,B 0,C 180,E1 -11527.255,E2 -11527.255} C_VEL
LIN {X 0,Y 390.015,Z 872.612,A -85,B 0,C 180,E1 -11528.812,E2 -11528.812} C_VEL
LIN {X 0,Y 390.612,Z 866.449,A -85,B 0,C 180,E1 -11530.366,E2 -11530.366} C_VEL
LIN {X 0,Y 391.435,Z 858.792,A -85,B 0,C 180,E1 -11531.917,E2 -11531.917} C_VEL
LIN {X 0,Y 392.136,Z 851.031,A -85,B 0,C 180,E1 -11533.21,E2 -11533.21} C_VEL
LIN {X 0,Y 393.089,Z 841.618,A -85,B 0,C 180,E1 -11534.496,E2 -11534.496} C_VEL
LIN {X 0,Y 394.099,Z 829.905,A -85,B 0,C 180,E1 -11535.782,E2 -11535.782} C_VEL
LIN {X 0,Y 395.127,Z 818.196,A -85,B 0,C 180,E1 -11536.801,E2 -11536.801} C_VEL
LIN {X 0,Y 395.816,Z 809.175,A -85,B 0,C 180,E1 -11537.436,E2 -11537.436} C_VEL
LIN {X 0,Y 394.221,Z 801.034,A -85,B 0,C 180,E1 -11538.048,E2 -11538.048} C_VEL
LIN {X 0,Y 390.355,Z 788.712,A -85,B 0,C 180,E1 -11538.927,E2 -11538.927} C_VEL
LIN {X 0,Y 389.42,Z 785.871,A -85,B 0,C 180,E1 -11539.129,E2 -11539.129} C_VEL
LIN {X 0,Y 389.479,Z 781.868,A -85,B 0,C 180,E1 -11543.033,E2 -11543.033} C_VEL
LIN {X 0,Y 389.56,Z 777.934,A -85,B 0,C 180,E1 -11546.81,E2 -11546.81} C_VEL
LIN {X 0,Y 389.607,Z 774.19,A -85,B 0,C 180,E1 -11550.338,E2 -11550.338} C_VEL
LIN {X 0,Y 389.577,Z 772.967,A -85,B 0,C 180,E1 -11551.546,E2 -11551.546} C_VEL
LIN {X 0,Y 389.875,Z 772.923,A -85,B 0,C 180,E1 -11553.982,E2 -11553.982} C_VEL
LIN {X 0,Y 390.009,Z 772.905,A -85,B 0,C 180,E1 -11556.49,E2 -11556.49} C_VEL
LIN {X 0,Y 390.065,Z 772.898,A -85,B 0,C 180,E1 -11559.217,E2 -11559.217} C_VEL
LIN {X 0,Y 390.043,Z 772.899,A -85,B 0,C 180,E1 -11562.374,E2 -11562.374} C_VEL
LIN {X 0,Y 390.04,Z 772.901,A -85,B 0,C 180,E1 -11565.777,E2 -11565.777} C_VEL
LIN {X 0,Y 390.06,Z 772.949,A -85,B 0,C 180,E1 -11566.114,E2 -11566.114} C_VEL
LIN {X 0,Y 391.008,Z 778.179,A -85,B 0,C 180,E1 -11569.019,E2 -11569.019} C_VEL
LIN {X 0,Y 392.144,Z 784.673,A -85,B 0,C 180,E1 -11572.457,E2 -11572.457} C_VEL
LIN {X 0,Y 392.349,Z 788.546,A -85,B 0,C 180,E1 -11574.397,E2 -11574.397} C_VEL
LIN {X 0,Y 391.74,Z 795.031,A -85,B 0,C 180,E1 -11577.481,E2 -11577.481} C_VEL
LIN {X 0,Y 391.138,Z 801.325,A -85,B 0,C 180,E1 -11580.388,E2 -11580.388} C_VEL
LIN {X 0,Y 390.641,Z 807.701,A -85,B 0,C 180,E1 -11583.271,E2 -11583.271} C_VEL
LIN {X 0,Y 390.031,Z 815.629,A -85,B 0,C 180,E1 -11586.778,E2 -11586.778} C_VEL
LIN {X 0,Y 389.662,Z 822.961,A -85,B 0,C 180,E1 -11589.959,E2 -11589.959} C_VEL
LIN {X 0,Y 389.471,Z 826.051,A -85,B 0,C 180,E1 -11591.251,E2 -11591.251} C_VEL
